// TIA Portal V15.1 export
// export: Created 2024-06-21T08:40:56.7100426Z, ExportSetting WithDefaults, DisplayName Totally Integrated Automation Portal, DisplayVersion V15.1 Update 5, DisplayName TIA Portal Openness, DisplayVersion V15.1 Update 5, DisplayName SINAMICS Startdrive Advanced, DisplayVersion V15.1, DisplayName G130, G150, S120, S150, SINAMICS MV, S210, DisplayVersion V15.1, DisplayName G110M, G120, G120C, G120D, G120P, DisplayVersion V15.1, DisplayName STEP 7 Professional, DisplayVersion V15.1 Update 5, DisplayName STEP 7 Safety, DisplayVersion V15.1, DisplayName WinCC Professional, DisplayVersion V15.1 Update 5, DisplayName SIMATIC Visualization Architect, DisplayVersion V15.1
FUNCTION_BLOCK "L3StopPos"   // FB2188, FBD
TITLE = L3StopPos
{ S7_Optimized_Access := 'TRUE' }
AUTHOR : VCC
FAMILY : Actuator
VERSION : 0.1
// =============================================================================
// This module will be used for a three Position movements.
// It will take care of the Alarms and of the Detections.
// =============================================================================
// stored: AutoNumber false, IsIECCheckEnabled false, IsRetainMemResEnabled false, MemoryReserve 100, SetENOAutomatically False, UDAEnableTagReadback false
   VAR_INPUT
      I_DetPos1 { ExternalAccessible := 'False'; ExternalVisible := 'False'; ExternalWritable := 'False'} : Bool;   // Set detection signal / Pos1 Detection signal
      I_DetPos2 { ExternalAccessible := 'False'; ExternalVisible := 'False'; ExternalWritable := 'False'} : Bool;   // Set detection signal / Pos2 Detection signal
      I_DetPos3 { ExternalAccessible := 'False'; ExternalVisible := 'False'; ExternalWritable := 'False'} : Bool;   // Reset detection signal / Pos3 Detection signal
      I_CmdPos1 { ExternalAccessible := 'False'; ExternalVisible := 'False'; ExternalWritable := 'False'} : Bool;   // function set command / Function Pos1 command
      I_CmdPos2 { ExternalAccessible := 'False'; ExternalVisible := 'False'; ExternalWritable := 'False'} : Bool;   // function set command / Function Pos2 command
      I_CmdPos3 { ExternalAccessible := 'False'; ExternalVisible := 'False'; ExternalWritable := 'False'} : Bool;   // Function reset command / Function Pos3 command
      I_RunPos1 { ExternalAccessible := 'False'; ExternalVisible := 'False'; ExternalWritable := 'False'} : Bool;   // Memory that the Set function is busy / Memory that the Pos1 function is busy
      I_RunPos2 { ExternalAccessible := 'False'; ExternalVisible := 'False'; ExternalWritable := 'False'} : Bool;   // Memory that the Set function is busy / Memory that the Pos2 function is busy
      I_RunPos3 { ExternalAccessible := 'False'; ExternalVisible := 'False'; ExternalWritable := 'False'} : Bool;   // Memory that the Reset function is busy / Memory that the Pos3 function is busy
      I_Pos1IntlkOK { ExternalAccessible := 'False'; ExternalVisible := 'False'; ExternalWritable := 'False'} : Bool;   // Set Interlock / Pos1 Interlock
      I_Pos2IntlkOK { ExternalAccessible := 'False'; ExternalVisible := 'False'; ExternalWritable := 'False'} : Bool;   // Set Interlock / Pos2 Interlock
      I_Pos3IntlkOK { ExternalAccessible := 'False'; ExternalVisible := 'False'; ExternalWritable := 'False'} : Bool;   // Reset Interlock / Pos3 Interlock
      I_SafetyOk { ExternalAccessible := 'False'; ExternalVisible := 'False'; ExternalWritable := 'False'} : Bool;   // Safety Ok
      I_AlarmResetPB { ExternalAccessible := 'False'; ExternalVisible := 'False'; ExternalWritable := 'False'} : Bool := TRUE;   // alarm reset Push Button is activated / Alarm Reset Push Button is Activated
      C_KeepPosition { ExternalAccessible := 'False'; ExternalVisible := 'False'; ExternalWritable := 'False'} : Bool;   // If true, the last position shall be kept ON and checked / If true, the last Position shall be kept ON and checked
      C_EnAlmDet { ExternalAccessible := 'False'; ExternalVisible := 'False'; ExternalWritable := 'False'} : Bool;   // Enable alarm / Enable Alarm
      C_AlarmResetUsed { ExternalAccessible := 'False'; ExternalVisible := 'False'; ExternalWritable := 'False'} : Bool;   // If true, the alarms will be stored untill reseted / If true, the Alarms will be stored untill Reseted
      C_EnAlmOvertime { ExternalAccessible := 'False'; ExternalVisible := 'False'; ExternalWritable := 'False'} : Bool := TRUE;   // Enable Overtime Alarm
      C_RunTimeMaxPos1Warn { ExternalAccessible := 'False'; ExternalVisible := 'False'; ExternalWritable := 'False'} : DInt;   // Maximum Time (ms) that the function may run (create overtime) / Maximum Time (ms) that the function may run (create Overtime)
      C_RunTimeMaxPos1Alm { ExternalAccessible := 'False'; ExternalVisible := 'False'; ExternalWritable := 'False'} : DInt;   // Maximum Time (ms) that the function may run (create overtime) / Maximum Time (ms) that the function may run (create Overtime)
      C_RunTimeMaxPos2Warn { ExternalAccessible := 'False'; ExternalVisible := 'False'; ExternalWritable := 'False'} : DInt;   // Maximum Time (ms) that the function may run (create overtime) / Maximum Time (ms) that the function may run (create Overtime)
      C_RunTimeMaxPos2Alm { ExternalAccessible := 'False'; ExternalVisible := 'False'; ExternalWritable := 'False'} : DInt;   // Maximum Time (ms) that the function may run (create overtime) / Maximum Time (ms) that the function may run (create Overtime)
      C_RunTimeMaxPos3Warn { ExternalAccessible := 'False'; ExternalVisible := 'False'; ExternalWritable := 'False'} : DInt;   // Maximum Time (ms) that the function may run (create overtime) / Maximum Time (ms) that the function may run (create Overtime)
      C_RunTimeMaxPos3Alm { ExternalAccessible := 'False'; ExternalVisible := 'False'; ExternalWritable := 'False'} : DInt;   // Maximum Time (ms) that the function may run (create overtime) / Maximum Time (ms) that the function may run (create Overtime)
      C_TimeAlmFilt { ExternalAccessible := 'False'; ExternalVisible := 'False'; ExternalWritable := 'False'} : DInt := L#2000;   // timer before any actuator alarm will be active (welding..) / timer before any actuator Alarm will be active (welding..)
      C_AlarmSeverityAB { ExternalAccessible := 'False'; ExternalVisible := 'False'; ExternalWritable := 'False'} : Bool;   // Alarm severity
   END_VAR
   VAR_OUTPUT
      O_Pos1 { ExternalAccessible := 'False'; ExternalVisible := 'False'; ExternalWritable := 'False'} : Bool;   // Actuator is in set position / Actuator is in Pos1 Position
      O_Pos2 { ExternalAccessible := 'False'; ExternalVisible := 'False'; ExternalWritable := 'False'} : Bool;   // Actuator is in reset position / Actuator is in Pos2 Position
      O_Pos3 { ExternalAccessible := 'False'; ExternalVisible := 'False'; ExternalWritable := 'False'} : Bool;   // Actuator is in reset position / Actuator is in Pos3 Position
      O_KeepPosPos1Alm { ExternalAccessible := 'False'; ExternalVisible := 'False'; ExternalWritable := 'False'} : Bool;   // Detection Set alarm / Detection Pos1 Alarm
      O_KeepPosPos2Alm { ExternalAccessible := 'False'; ExternalVisible := 'False'; ExternalWritable := 'False'} : Bool;   // Detection Reset alarm / Detection Pos2 Alarm
      O_KeepPosPos3Alm { ExternalAccessible := 'False'; ExternalVisible := 'False'; ExternalWritable := 'False'} : Bool;   // Detection Reset alarm / Detection Pos3 Alarm
      O_MoreThenOneDetAlm { ExternalAccessible := 'False'; ExternalVisible := 'False'; ExternalWritable := 'False'} : Bool;   // Fault condition Both detections ON at the same time / Fault condition More Than One Detections On at the same time
      O_OvtPos1Warn { ExternalAccessible := 'False'; ExternalVisible := 'False'; ExternalWritable := 'False'} : Bool;   // Warning Overtime Set / Warning Overtime Pos1
      O_OvtPos2Warn { ExternalAccessible := 'False'; ExternalVisible := 'False'; ExternalWritable := 'False'} : Bool;   // Warning Overtime Set / Warning Overtime Pos2
      O_OvtPos3Warn { ExternalAccessible := 'False'; ExternalVisible := 'False'; ExternalWritable := 'False'} : Bool;   // Warning Overtime Reset / Warning Overtime Pos3
      O_OvtPos1Alm { ExternalAccessible := 'False'; ExternalVisible := 'False'; ExternalWritable := 'False'} : Bool;   // Alarm Overtime Set / Alarm Overtime Pos1
      O_OvtPos2Alm { ExternalAccessible := 'False'; ExternalVisible := 'False'; ExternalWritable := 'False'} : Bool;   // Alarm Overtime Set / Alarm Overtime Pos2
      O_OvtPos3Alm { ExternalAccessible := 'False'; ExternalVisible := 'False'; ExternalWritable := 'False'} : Bool;   // Alarm Overtime Reset / Alarm Overtime Pos3
      O_ConfigCalibrationAlm { ExternalAccessible := 'False'; ExternalVisible := 'False'; ExternalWritable := 'False'} : Bool;   // Alarm Config/Calibration
      O_CalibrationWarn { ExternalAccessible := 'False'; ExternalVisible := 'False'; ExternalWritable := 'False'} : Bool;   // Warning Calibration
      O_AlarmABCondition { ExternalAccessible := 'False'; ExternalVisible := 'False'; ExternalWritable := 'False'} : Bool;   // Alarm AB condition / Alarm AB Condition
      H_IAnim { ExternalAccessible := 'False'; ExternalVisible := 'False'; ExternalWritable := 'False'} : DWord;   // Icon animation Word / Icon Animation
   END_VAR
   VAR_IN_OUT
      IO_Modes : "Modes";   // Modes
      H_3StopPos : "H_3StopPos";   // Animation
   END_VAR
   VAR
      AlarmReset { ExternalAccessible := 'False'; ExternalVisible := 'False'; ExternalWritable := 'False'} : Bool;   // Alarm Reset Memory
      Pos1PosReq { ExternalAccessible := 'False'; ExternalVisible := 'False'; ExternalWritable := 'False'} : Bool;   // Memorisation of the last set movement / Memorisation of the last Pos1 movement
      Pos2PosReq { ExternalAccessible := 'False'; ExternalVisible := 'False'; ExternalWritable := 'False'} : Bool;   // Memorisation of the last reset movement / Memorisation of the last Pos2 movement
      Pos3PosReq { ExternalAccessible := 'False'; ExternalVisible := 'False'; ExternalWritable := 'False'} : Bool;   // Memorisation of the last reset movement / Memorisation of the last Pos3 movement
      KeepPos1PosOn { ExternalAccessible := 'False'; ExternalVisible := 'False'; ExternalWritable := 'False'} : Bool;   // Check that Set detection is keept on / Check that Pos1 Detection is keept on
      KeepPos2PosOn { ExternalAccessible := 'False'; ExternalVisible := 'False'; ExternalWritable := 'False'} : Bool;   // Check that Set detection is keept on / Check that Pos2 Detection is keept on
      KeepPos3PosOn { ExternalAccessible := 'False'; ExternalVisible := 'False'; ExternalWritable := 'False'} : Bool;   // Check that Set detection is keept on / Check that Pos3 Detection is keept on
      KeepPosPos1StartTimer { ExternalAccessible := 'False'; ExternalVisible := 'False'; ExternalWritable := 'False'} : Bool;   // Detection Set request to start timer / Detection Pos1 Request to start timer
      KeepPosPos2StartTimer { ExternalAccessible := 'False'; ExternalVisible := 'False'; ExternalWritable := 'False'} : Bool;   // Detection Reset request to start timer / Detection Pos2 Request to start timer
      KeepPosPos3StartTimer { ExternalAccessible := 'False'; ExternalVisible := 'False'; ExternalWritable := 'False'} : Bool;   // Detection Reset request to start timer / Detection Pos3 Request to start timer
      MoreThenOneDet { ExternalAccessible := 'False'; ExternalVisible := 'False'; ExternalWritable := 'False'} : Bool;   // Both detections ON at the same time request to start timer / Both Detections ON at the same time Request to start timer
      AlarmFilterStart { ExternalAccessible := 'False'; ExternalVisible := 'False'; ExternalWritable := 'False'} : Bool;   // Alarm filter must be started
      OvtPos1WarnResult { ExternalAccessible := 'False'; ExternalVisible := 'False'; ExternalWritable := 'False'} : Bool;   // Overtime set warning result / Overtime Pos1 warning result
      OvtPos2WarnResult { ExternalAccessible := 'False'; ExternalVisible := 'False'; ExternalWritable := 'False'} : Bool;   // Overtime set warning result / Overtime Pos2 warning result
      OvtPos3WarnResult { ExternalAccessible := 'False'; ExternalVisible := 'False'; ExternalWritable := 'False'} : Bool;   // Overtime reset warning result / Overtime Pos3 warning result
      OvtPos1AlmResult { ExternalAccessible := 'False'; ExternalVisible := 'False'; ExternalWritable := 'False'} : Bool;   // Overtime set alarm result / Overtime Pos1 Alarm result
      OvtPos2AlmResult { ExternalAccessible := 'False'; ExternalVisible := 'False'; ExternalWritable := 'False'} : Bool;   // Overtime reset alarm result / Overtime Pos2 Alarm result
      OvtPos3AlmResult { ExternalAccessible := 'False'; ExternalVisible := 'False'; ExternalWritable := 'False'} : Bool;   // Overtime reset alarm result / Overtime Pos3 Alarm result
      AlmFilterResult { ExternalAccessible := 'False'; ExternalVisible := 'False'; ExternalWritable := 'False'} : Bool;   // Alarm filter result
      MoreThenOneDetAlm { ExternalAccessible := 'False'; ExternalVisible := 'False'; ExternalWritable := 'False'} : Bool;   // Two detection alarm / Pos1 Pos2 Pos3 More Than One Activated
      KeepPos3Alm { ExternalAccessible := 'False'; ExternalVisible := 'False'; ExternalWritable := 'False'} : Bool;   // Keep position Reset alarm / Alarm Keep Position Pos3 Position / Larm Positionsövervakning Pos3 Läge
      KeepPos2Alm { ExternalAccessible := 'False'; ExternalVisible := 'False'; ExternalWritable := 'False'} : Bool;   // Keep position Set alarm / Alarm Keep Position Pos2 Position / Larm Positionsövervakning Pos2 Läge
      KeepPos1Alm { ExternalAccessible := 'False'; ExternalVisible := 'False'; ExternalWritable := 'False'} : Bool;   // Keep position Set alarm / Alarm Keep Position Pos1 Position / Larm Positionsövervakning Pos1 Läge
      OvtPos3Alm { ExternalAccessible := 'False'; ExternalVisible := 'False'; ExternalWritable := 'False'} : Bool;   // Overtime Reset alarm / Overtime Pos3 Alarm
      OvtPos2Alm { ExternalAccessible := 'False'; ExternalVisible := 'False'; ExternalWritable := 'False'} : Bool;   // Overtime Set alarm / Overtime Pos2 Alarm
      OvtPos1Alm { ExternalAccessible := 'False'; ExternalVisible := 'False'; ExternalWritable := 'False'} : Bool;   // Overtime Set alarm / Overtime Pos1 Alarm
      OvtPos3Warn { ExternalAccessible := 'False'; ExternalVisible := 'False'; ExternalWritable := 'False'} : Bool;   // Overtime Reset warning / Overtime Pos3 warning
      OvtPos2Warn { ExternalAccessible := 'False'; ExternalVisible := 'False'; ExternalWritable := 'False'} : Bool;   // Overtime Reset warning / Overtime Pos2 warning
      OvtPos1Warn { ExternalAccessible := 'False'; ExternalVisible := 'False'; ExternalWritable := 'False'} : Bool;   // Overtime Set warning / Overtime Pos1 warning
      ConfigCalibrationAlm { ExternalAccessible := 'False'; ExternalVisible := 'False'; ExternalWritable := 'False'} : Bool;   // Config/Calibration Alarm
      CalibrationWarn { ExternalAccessible := 'False'; ExternalVisible := 'False'; ExternalWritable := 'False'} : Bool;   // Warning Calibration
      Pos1Pos { ExternalAccessible := 'False'; ExternalVisible := 'False'; ExternalWritable := 'False'} : Bool;   // Set position / Pos1 Position
      Pos2Pos { ExternalAccessible := 'False'; ExternalVisible := 'False'; ExternalWritable := 'False'} : Bool;   // Set position / Pos2 Position
      Pos3Pos { ExternalAccessible := 'False'; ExternalVisible := 'False'; ExternalWritable := 'False'} : Bool;   // Reset position / Pos3 Position
      KeepPosPos3AlmCond { ExternalAccessible := 'False'; ExternalVisible := 'False'; ExternalWritable := 'False'} : Bool;   // Keep position reset alarm condition / Keep Position Pos3 Alarm condition
      KeepPosPos2AlmCond { ExternalAccessible := 'False'; ExternalVisible := 'False'; ExternalWritable := 'False'} : Bool;   // Keep position set alarm condition / Keep Position Pos1 Alarm condition
      KeepPosPos1AlmCond { ExternalAccessible := 'False'; ExternalVisible := 'False'; ExternalWritable := 'False'} : Bool;   // Keep position set alarm condition / Keep Position Pos1 Alarm condition
      TwoDetAlmCond { ExternalAccessible := 'False'; ExternalVisible := 'False'; ExternalWritable := 'False'} : Bool;   // Two detector alarm condition / Two or More Detection Alarm condition
      OvtPos3AlmCond { ExternalAccessible := 'False'; ExternalVisible := 'False'; ExternalWritable := 'False'} : Bool;   // Overtime reset alarm condition / Overtime Pos3 Alarm condition
      OvtPos2AlmCond { ExternalAccessible := 'False'; ExternalVisible := 'False'; ExternalWritable := 'False'} : Bool;   // Overtime reset alarm condition / Overtime Pos2 Alarm condition
      OvtPos1AlmCond { ExternalAccessible := 'False'; ExternalVisible := 'False'; ExternalWritable := 'False'} : Bool;   // Overtime set alarm condition / Overtime Pos1 Alarm condition
      Edge { ExternalAccessible := 'False'; ExternalVisible := 'False'; ExternalWritable := 'False'} : Array[1..8] of Bool;   // Edge
      AlarmTimer { ExternalAccessible := 'False'; ExternalVisible := 'False'; ExternalWritable := 'False'} : "LTimer";   // FB
      OvtPos1WarnTimer { ExternalAccessible := 'False'; ExternalVisible := 'False'; ExternalWritable := 'False'} : "LTimer";   // FB
      OvtPos2WarnTimer { ExternalAccessible := 'False'; ExternalVisible := 'False'; ExternalWritable := 'False'} : "LTimer";   // FB
      OvtPos3WarnTimer { ExternalAccessible := 'False'; ExternalVisible := 'False'; ExternalWritable := 'False'} : "LTimer";   // FB
      OvtPos1AlmTimer { ExternalAccessible := 'False'; ExternalVisible := 'False'; ExternalWritable := 'False'} : "LTimer";   // FB
      OvtPos2AlmTimer { ExternalAccessible := 'False'; ExternalVisible := 'False'; ExternalWritable := 'False'} : "LTimer";   // FB
      OvtPos3AlmTimer { ExternalAccessible := 'False'; ExternalVisible := 'False'; ExternalWritable := 'False'} : "LTimer";   // FB
   END_VAR
   VAR RETAIN
      OvtWarnPos1 { ExternalAccessible := 'False'; ExternalVisible := 'False'; ExternalWritable := 'False'} : DInt;   // Alarm Value
      OvtWarnPos2 { ExternalAccessible := 'False'; ExternalVisible := 'False'; ExternalWritable := 'False'} : DInt;   // Alarm Value
      OvtWarnPos3 { ExternalAccessible := 'False'; ExternalVisible := 'False'; ExternalWritable := 'False'} : DInt;   // Alarm Value
      OvtWarnPos1toPos2 { ExternalAccessible := 'False'; ExternalVisible := 'False'; ExternalWritable := 'False'} : DInt;   // Alarm Value
      OvtWarnPos1toPos3 { ExternalAccessible := 'False'; ExternalVisible := 'False'; ExternalWritable := 'False'} : DInt;   // Alarm Value
      OvtWarnPos2toPos3 { ExternalAccessible := 'False'; ExternalVisible := 'False'; ExternalWritable := 'False'} : DInt;   // Alarm Value
      OvtWarnPos2toPos1 { ExternalAccessible := 'False'; ExternalVisible := 'False'; ExternalWritable := 'False'} : DInt;   // Alarm Value
      OvtWarnPos3toPos2 { ExternalAccessible := 'False'; ExternalVisible := 'False'; ExternalWritable := 'False'} : DInt;   // Alarm Value
      OvtWarnPos3toPos1 { ExternalAccessible := 'False'; ExternalVisible := 'False'; ExternalWritable := 'False'} : DInt;   // Alarm Value
      OvtAlarmPos1 { ExternalAccessible := 'False'; ExternalVisible := 'False'; ExternalWritable := 'False'} : DInt;   // Alarm Value
      OvtAlarmPos2 { ExternalAccessible := 'False'; ExternalVisible := 'False'; ExternalWritable := 'False'} : DInt;   // Alarm Value
      OvtAlarmPos3 { ExternalAccessible := 'False'; ExternalVisible := 'False'; ExternalWritable := 'False'} : DInt;   // Alarm Value
      OvtAlarmPos1toPos2 { ExternalAccessible := 'False'; ExternalVisible := 'False'; ExternalWritable := 'False'} : DInt;   // Alarm Value
      OvtAlarmPos1toPos3 { ExternalAccessible := 'False'; ExternalVisible := 'False'; ExternalWritable := 'False'} : DInt;   // Alarm Value
      OvtAlarmPos2toPos3 { ExternalAccessible := 'False'; ExternalVisible := 'False'; ExternalWritable := 'False'} : DInt;   // Alarm Value
      OvtAlarmPos2toPos1 { ExternalAccessible := 'False'; ExternalVisible := 'False'; ExternalWritable := 'False'} : DInt;   // Alarm Value
      OvtAlarmPos3toPos2 { ExternalAccessible := 'False'; ExternalVisible := 'False'; ExternalWritable := 'False'} : DInt;   // Alarm Value
      OvtAlarmPos3toPos1 { ExternalAccessible := 'False'; ExternalVisible := 'False'; ExternalWritable := 'False'} : DInt;   // Alarm Value
      CalibratedPos1toPos2 { ExternalAccessible := 'False'; ExternalVisible := 'False'; ExternalWritable := 'False'} : Bool;   // Calibrated Set
      CalibratedPos1toPos3 { ExternalAccessible := 'False'; ExternalVisible := 'False'; ExternalWritable := 'False'} : Bool;   // Calibrated Reset
      CalibratedPos2toPos3 { ExternalAccessible := 'False'; ExternalVisible := 'False'; ExternalWritable := 'False'} : Bool;   // Calibrated Reset
      CalibratedPos2toPos1 { ExternalAccessible := 'False'; ExternalVisible := 'False'; ExternalWritable := 'False'} : Bool;   // Calibrated Reset
      CalibratedPos3toPos2 { ExternalAccessible := 'False'; ExternalVisible := 'False'; ExternalWritable := 'False'} : Bool;   // Calibrated Reset
      CalibratedPos3toPos1 { ExternalAccessible := 'False'; ExternalVisible := 'False'; ExternalWritable := 'False'} : Bool;   // Calibrated Reset
      MovementPos1toPos3 { ExternalAccessible := 'False'; ExternalVisible := 'False'; ExternalWritable := 'False'} : Bool;   // Calibrated Set
      MovementPos1toPos2 { ExternalAccessible := 'False'; ExternalVisible := 'False'; ExternalWritable := 'False'} : Bool;   // Calibrated Set
      MovementPos3toPos1 { ExternalAccessible := 'False'; ExternalVisible := 'False'; ExternalWritable := 'False'} : Bool;   // Calibrated Set
      MovementPos3toPos2 { ExternalAccessible := 'False'; ExternalVisible := 'False'; ExternalWritable := 'False'} : Bool;   // Calibrated Set
      MovementPos2toPos1 { ExternalAccessible := 'False'; ExternalVisible := 'False'; ExternalWritable := 'False'} : Bool;   // Calibrated Set
      MovementPos2toPos3 { ExternalAccessible := 'False'; ExternalVisible := 'False'; ExternalWritable := 'False'} : Bool;   // Calibrated Set
   END_VAR
   VAR
      AlarmTimeWithConfig { ExternalAccessible := 'False'; ExternalVisible := 'False'; ExternalWritable := 'False'} : Bool;
      AlarmTimeWithCalibration { ExternalAccessible := 'False'; ExternalVisible := 'False'; ExternalWritable := 'False'} : Bool;
      AlmFilterTimerValue { ExternalAccessible := 'False'; ExternalVisible := 'False'; ExternalWritable := 'False'} : DInt;
   END_VAR
   VAR_TEMP
      Cnt : Int;   // Temp
      H_CalibratePos1 : Bool;   // HMI Function
      H_CalibratePos2 : Bool;   // HMI Function
      H_CalibratePos3 : Bool;   // HMI Function
      TempReal : Real;
   END_VAR
   VAR_TEMP   // added for the SCL form of the ladder/FBD networks
      _w1 : Bool;
      _w2 : Bool;
      _w3 : Bool;
      _w4 : Bool;
      _w5 : Bool;
      _w6 : Bool;
      _w7 : Bool;
      _w8 : Bool;
      _w9 : Bool;
      _w10 : Bool;
      _w11 : Bool;
      _w12 : Bool;
      _w13 : Bool;
      _w14 : Bool;
      _w15 : Bool;
   END_VAR
BEGIN

REGION Network 1: **** 1 - Inputs **** HMI Commands
   // Extract the Commands from HMIRobCmd / Extract the Commands from HMI
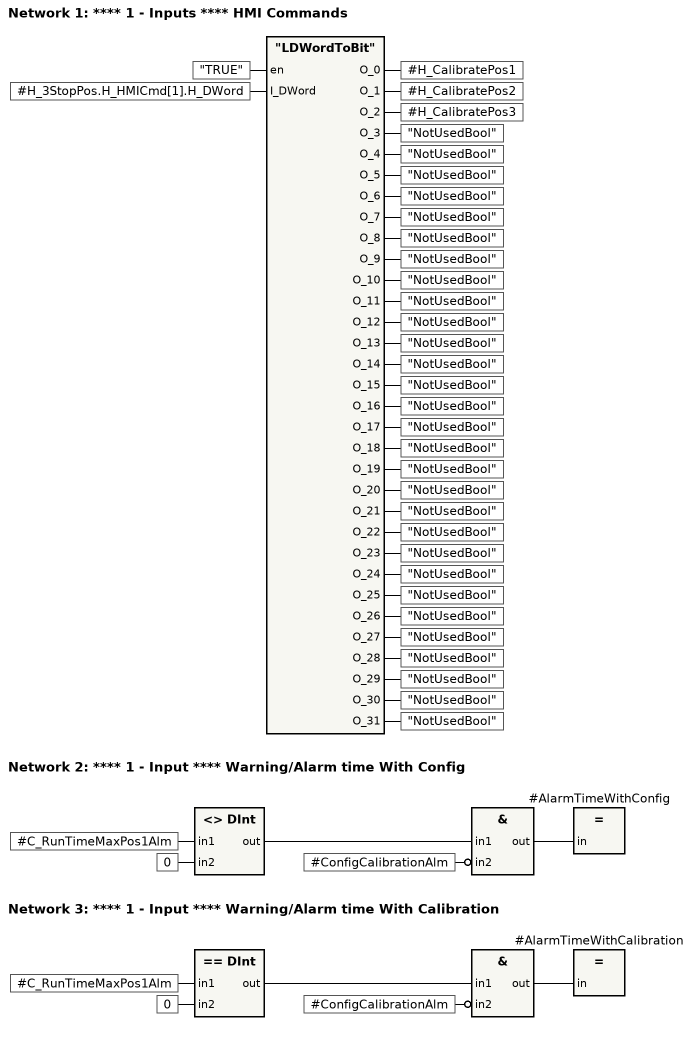
   IF "TRUE" THEN
       "LDWordToBit"(I_DWord := #H_3StopPos.H_HMICmd[1].H_DWord,
                     O_0 => #H_CalibratePos1,
                     O_1 => #H_CalibratePos2,
                     O_2 => #H_CalibratePos3,
                     O_3 => "NotUsedBool",
                     O_4 => "NotUsedBool",
                     O_5 => "NotUsedBool",
                     O_6 => "NotUsedBool",
                     O_7 => "NotUsedBool",
                     O_8 => "NotUsedBool",
                     O_9 => "NotUsedBool",
                     O_10 => "NotUsedBool",
                     O_11 => "NotUsedBool",
                     O_12 => "NotUsedBool",
                     O_13 => "NotUsedBool",
                     O_14 => "NotUsedBool",
                     O_15 => "NotUsedBool",
                     O_16 => "NotUsedBool",
                     O_17 => "NotUsedBool",
                     O_18 => "NotUsedBool",
                     O_19 => "NotUsedBool",
                     O_20 => "NotUsedBool",
                     O_21 => "NotUsedBool",
                     O_22 => "NotUsedBool",
                     O_23 => "NotUsedBool",
                     O_24 => "NotUsedBool",
                     O_25 => "NotUsedBool",
                     O_26 => "NotUsedBool",
                     O_27 => "NotUsedBool",
                     O_28 => "NotUsedBool",
                     O_29 => "NotUsedBool",
                     O_30 => "NotUsedBool",
                     O_31 => "NotUsedBool");
   END_IF;
END_REGION

REGION Network 2: **** 1 - Input **** Warning/Alarm time With Config
   #AlarmTimeWithConfig := (#C_RunTimeMaxPos1Alm <> 0) AND NOT #ConfigCalibrationAlm;
END_REGION

REGION Network 3: **** 1 - Input **** Warning/Alarm time With Calibration
   #AlarmTimeWithCalibration := (#C_RunTimeMaxPos1Alm = 0) AND NOT #ConfigCalibrationAlm;
END_REGION

REGION Network 4: Calibrated Set / **** 1 - Input **** Ovt Values / **** 1 - Inputs **** Ovt Values
   // Ovt Values
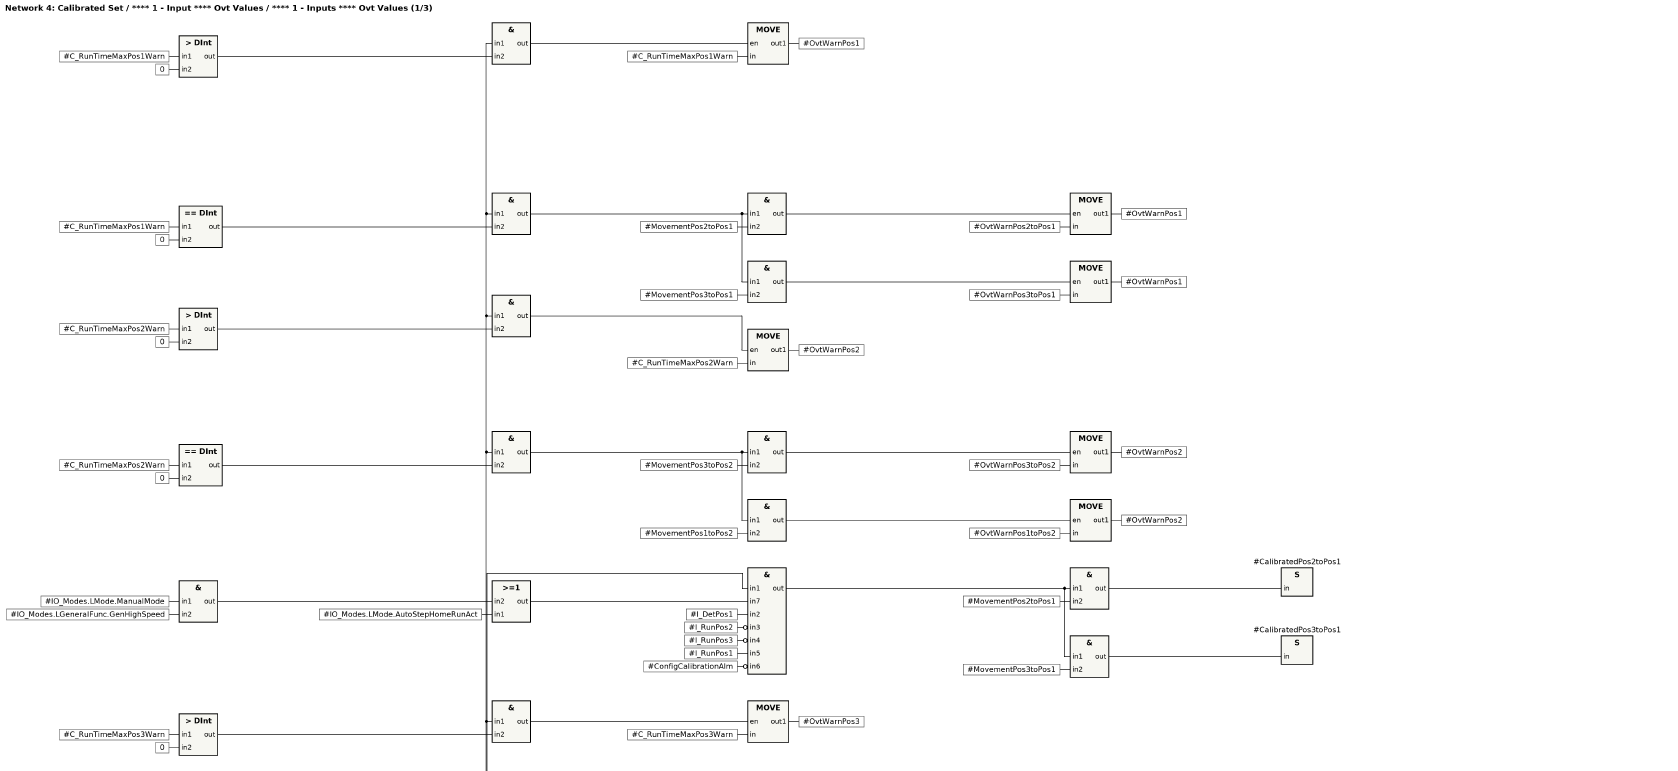
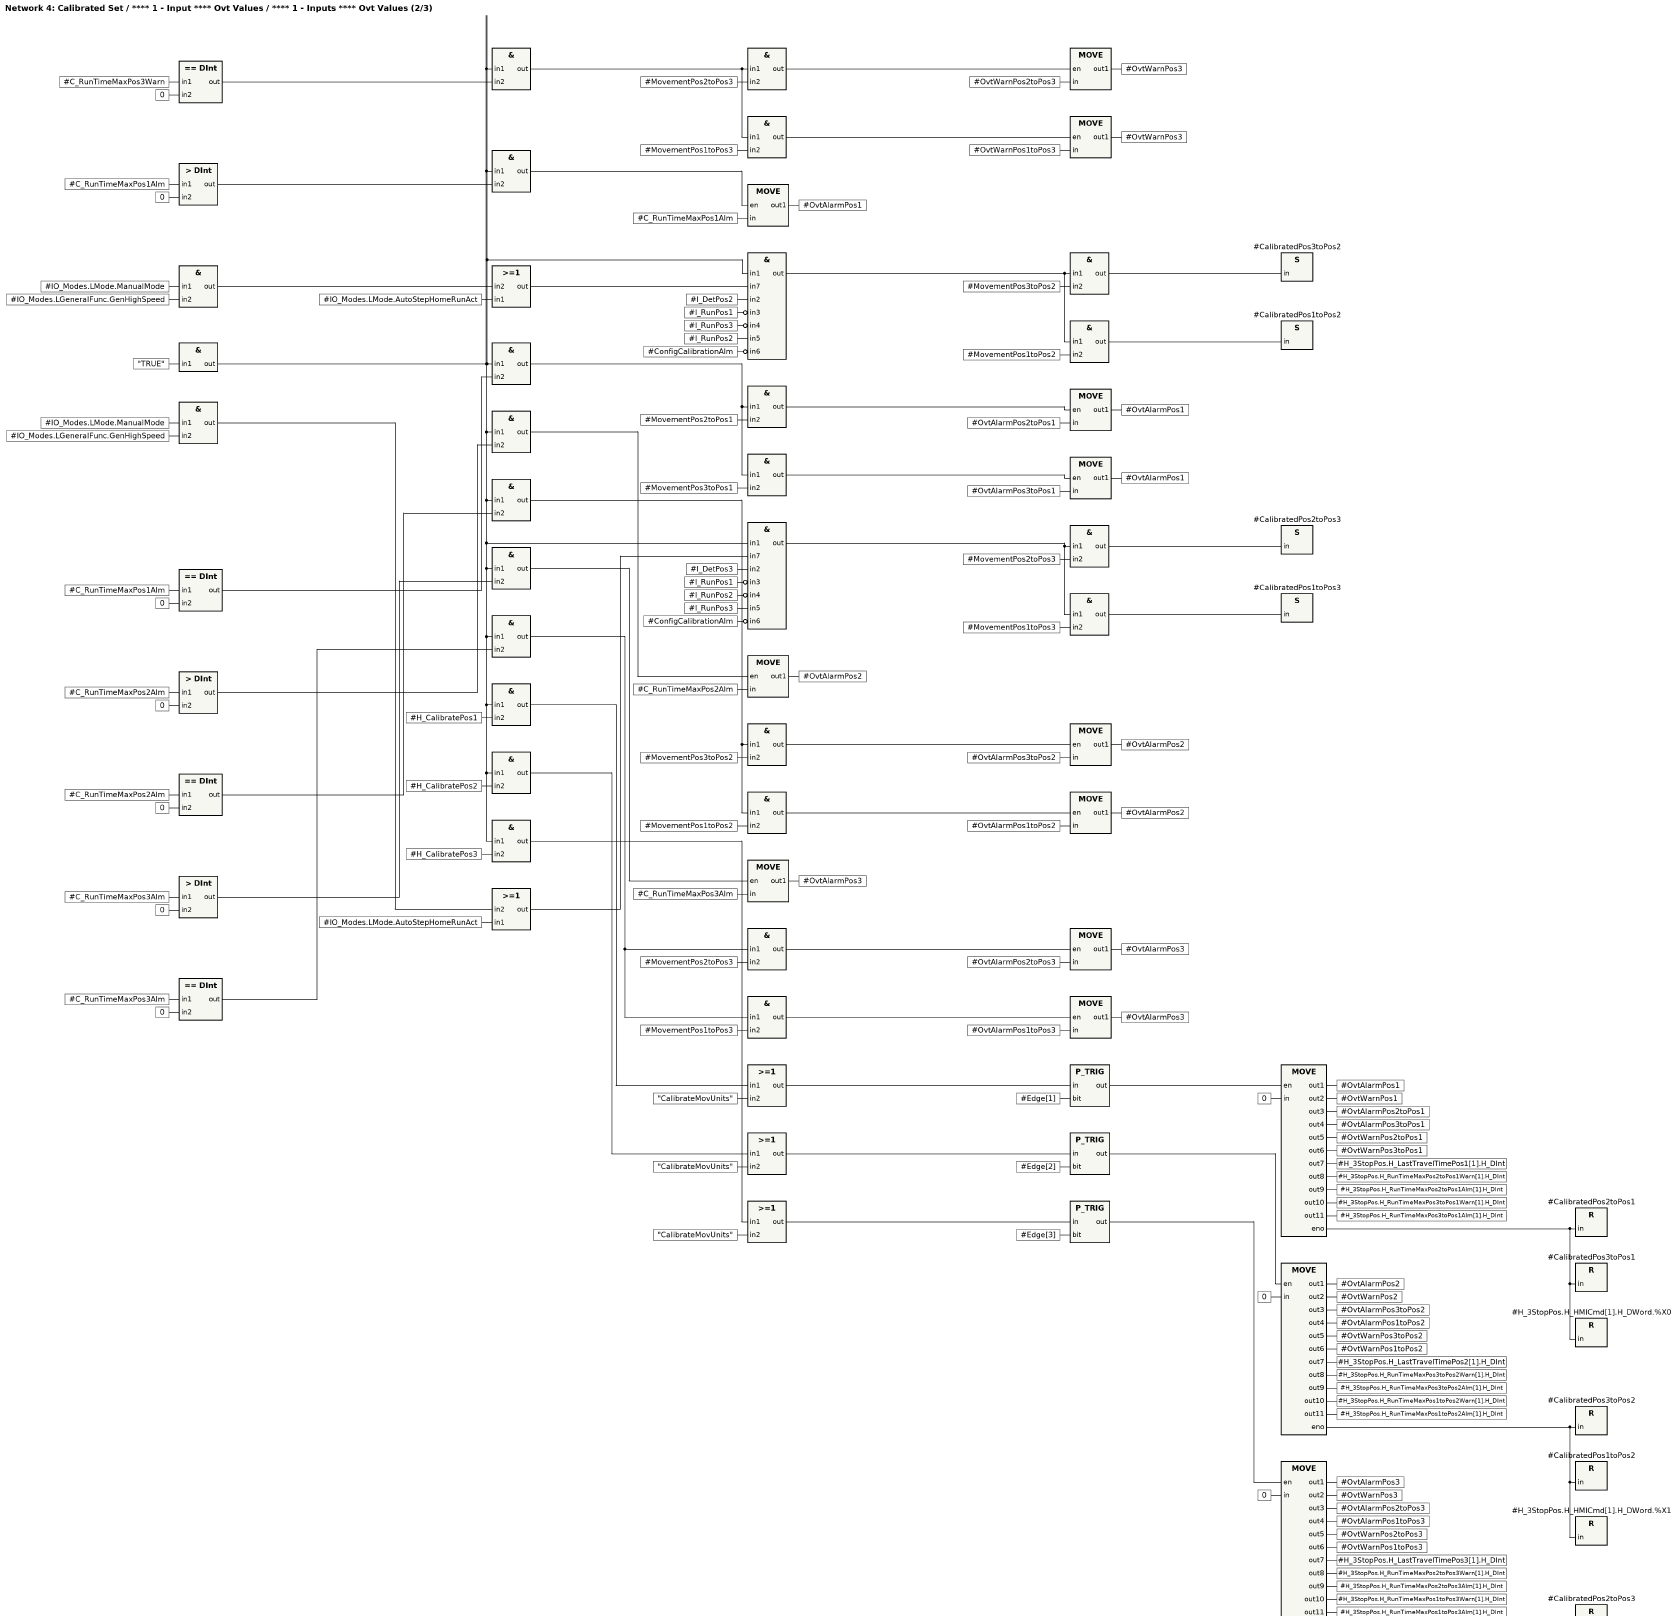
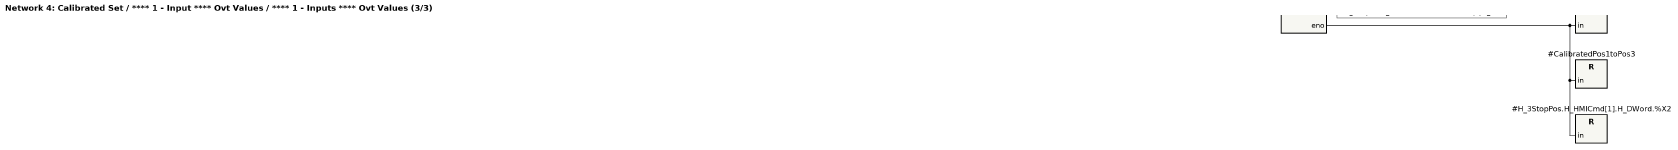
   // ENO of a box is taken as its EN; it also drops when the box reports an error
   IF "TRUE" AND (#C_RunTimeMaxPos1Warn > 0) THEN #OvtWarnPos1 := #C_RunTimeMaxPos1Warn; END_IF;
   #_w1 := "TRUE" AND (#C_RunTimeMaxPos1Warn = 0);
   IF #_w1 AND #MovementPos2toPos1 THEN #OvtWarnPos1 := #OvtWarnPos2toPos1; END_IF;
   IF #_w1 AND #MovementPos3toPos1 THEN #OvtWarnPos1 := #OvtWarnPos3toPos1; END_IF;
   IF "TRUE" AND (#C_RunTimeMaxPos2Warn > 0) THEN #OvtWarnPos2 := #C_RunTimeMaxPos2Warn; END_IF;
   #_w2 := "TRUE" AND (#C_RunTimeMaxPos2Warn = 0);
   IF #_w2 AND #MovementPos3toPos2 THEN #OvtWarnPos2 := #OvtWarnPos3toPos2; END_IF;
   IF #_w2 AND #MovementPos1toPos2 THEN #OvtWarnPos2 := #OvtWarnPos1toPos2; END_IF;
   IF "TRUE" AND (#C_RunTimeMaxPos3Warn > 0) THEN #OvtWarnPos3 := #C_RunTimeMaxPos3Warn; END_IF;
   #_w3 := "TRUE" AND (#C_RunTimeMaxPos3Warn = 0);
   IF #_w3 AND #MovementPos2toPos3 THEN #OvtWarnPos3 := #OvtWarnPos2toPos3; END_IF;
   IF #_w3 AND #MovementPos1toPos3 THEN #OvtWarnPos3 := #OvtWarnPos1toPos3; END_IF;
   IF "TRUE" AND (#C_RunTimeMaxPos1Alm > 0) THEN #OvtAlarmPos1 := #C_RunTimeMaxPos1Alm; END_IF;
   #_w4 := "TRUE" AND (#C_RunTimeMaxPos1Alm = 0);
   IF #_w4 AND #MovementPos2toPos1 THEN #OvtAlarmPos1 := #OvtAlarmPos2toPos1; END_IF;
   IF #_w4 AND #MovementPos3toPos1 THEN #OvtAlarmPos1 := #OvtAlarmPos3toPos1; END_IF;
   IF "TRUE" AND (#C_RunTimeMaxPos2Alm > 0) THEN #OvtAlarmPos2 := #C_RunTimeMaxPos2Alm; END_IF;
   #_w5 := "TRUE" AND (#C_RunTimeMaxPos2Alm = 0);
   IF #_w5 AND #MovementPos3toPos2 THEN #OvtAlarmPos2 := #OvtAlarmPos3toPos2; END_IF;
   IF #_w5 AND #MovementPos1toPos2 THEN #OvtAlarmPos2 := #OvtAlarmPos1toPos2; END_IF;
   IF "TRUE" AND (#C_RunTimeMaxPos3Alm > 0) THEN #OvtAlarmPos3 := #C_RunTimeMaxPos3Alm; END_IF;
   #_w6 := "TRUE" AND (#C_RunTimeMaxPos3Alm = 0);
   IF #_w6 AND #MovementPos2toPos3 THEN #OvtAlarmPos3 := #OvtAlarmPos2toPos3; END_IF;
   IF #_w6 AND #MovementPos1toPos3 THEN #OvtAlarmPos3 := #OvtAlarmPos1toPos3; END_IF;
   #_w7 := "TRUE" AND ((#IO_Modes.LMode.ManualMode AND #IO_Modes.LGeneralFunc.GenHighSpeed) OR #IO_Modes.LMode.AutoStepHomeRunAct) AND #I_DetPos1 AND NOT #I_RunPos2 AND NOT #I_RunPos3 AND #I_RunPos1 AND NOT #ConfigCalibrationAlm;
   IF #_w7 AND #MovementPos2toPos1 THEN #CalibratedPos2toPos1 := TRUE; END_IF;
   IF #_w7 AND #MovementPos3toPos1 THEN #CalibratedPos3toPos1 := TRUE; END_IF;
   #_w8 := "TRUE" AND ((#IO_Modes.LMode.ManualMode AND #IO_Modes.LGeneralFunc.GenHighSpeed) OR #IO_Modes.LMode.AutoStepHomeRunAct) AND #I_DetPos2 AND NOT #I_RunPos1 AND NOT #I_RunPos3 AND #I_RunPos2 AND NOT #ConfigCalibrationAlm;
   IF #_w8 AND #MovementPos3toPos2 THEN #CalibratedPos3toPos2 := TRUE; END_IF;
   IF #_w8 AND #MovementPos1toPos2 THEN #CalibratedPos1toPos2 := TRUE; END_IF;
   #_w9 := "TRUE" AND ((#IO_Modes.LMode.ManualMode AND #IO_Modes.LGeneralFunc.GenHighSpeed) OR #IO_Modes.LMode.AutoStepHomeRunAct) AND #I_DetPos3 AND NOT #I_RunPos1 AND NOT #I_RunPos2 AND #I_RunPos3 AND NOT #ConfigCalibrationAlm;
   IF #_w9 AND #MovementPos2toPos3 THEN #CalibratedPos2toPos3 := TRUE; END_IF;
   IF #_w9 AND #MovementPos1toPos3 THEN #CalibratedPos1toPos3 := TRUE; END_IF;
   #_w10 := ("TRUE" AND #H_CalibratePos1) OR "CalibrateMovUnits";
   #_w11 := #_w10 AND NOT #Edge[1];   // rising edge
   #Edge[1] := #_w10;
   IF #_w11 THEN
       #OvtAlarmPos1 := 0;
       #OvtWarnPos1 := 0;
       #OvtAlarmPos2toPos1 := 0;
       #OvtAlarmPos3toPos1 := 0;
       #OvtWarnPos2toPos1 := 0;
       #OvtWarnPos3toPos1 := 0;
       #H_3StopPos.H_LastTravelTimePos1[1].H_DInt := 0;
       #H_3StopPos.H_RunTimeMaxPos2toPos1Warn[1].H_DInt := 0;
       #H_3StopPos.H_RunTimeMaxPos2toPos1Alm[1].H_DInt := 0;
       #H_3StopPos.H_RunTimeMaxPos3toPos1Warn[1].H_DInt := 0;
       #H_3StopPos.H_RunTimeMaxPos3toPos1Alm[1].H_DInt := 0;
       #CalibratedPos2toPos1 := FALSE;
       #CalibratedPos3toPos1 := FALSE;
       #H_3StopPos.H_HMICmd[1].H_DWord.%X0 := FALSE;
   END_IF;
   #_w12 := ("TRUE" AND #H_CalibratePos2) OR "CalibrateMovUnits";
   #_w13 := #_w12 AND NOT #Edge[2];   // rising edge
   #Edge[2] := #_w12;
   IF #_w13 THEN
       #OvtAlarmPos2 := 0;
       #OvtWarnPos2 := 0;
       #OvtAlarmPos3toPos2 := 0;
       #OvtAlarmPos1toPos2 := 0;
       #OvtWarnPos3toPos2 := 0;
       #OvtWarnPos1toPos2 := 0;
       #H_3StopPos.H_LastTravelTimePos2[1].H_DInt := 0;
       #H_3StopPos.H_RunTimeMaxPos3toPos2Warn[1].H_DInt := 0;
       #H_3StopPos.H_RunTimeMaxPos3toPos2Alm[1].H_DInt := 0;
       #H_3StopPos.H_RunTimeMaxPos1toPos2Warn[1].H_DInt := 0;
       #H_3StopPos.H_RunTimeMaxPos1toPos2Alm[1].H_DInt := 0;
       #CalibratedPos3toPos2 := FALSE;
       #CalibratedPos1toPos2 := FALSE;
       #H_3StopPos.H_HMICmd[1].H_DWord.%X1 := FALSE;
   END_IF;
   #_w14 := ("TRUE" AND #H_CalibratePos3) OR "CalibrateMovUnits";
   #_w15 := #_w14 AND NOT #Edge[3];   // rising edge
   #Edge[3] := #_w14;
   IF #_w15 THEN
       #OvtAlarmPos3 := 0;
       #OvtWarnPos3 := 0;
       #OvtAlarmPos2toPos3 := 0;
       #OvtAlarmPos1toPos3 := 0;
       #OvtWarnPos2toPos3 := 0;
       #OvtWarnPos1toPos3 := 0;
       #H_3StopPos.H_LastTravelTimePos3[1].H_DInt := 0;
       #H_3StopPos.H_RunTimeMaxPos2toPos3Warn[1].H_DInt := 0;
       #H_3StopPos.H_RunTimeMaxPos2toPos3Alm[1].H_DInt := 0;
       #H_3StopPos.H_RunTimeMaxPos1toPos3Warn[1].H_DInt := 0;
       #H_3StopPos.H_RunTimeMaxPos1toPos3Alm[1].H_DInt := 0;
       #CalibratedPos2toPos3 := FALSE;
       #CalibratedPos1toPos3 := FALSE;
       #H_3StopPos.H_HMICmd[1].H_DWord.%X2 := FALSE;
   END_IF;
END_REGION

REGION Network 5: **** 1 - Input **** Start Movement from Pos1 to Pos3
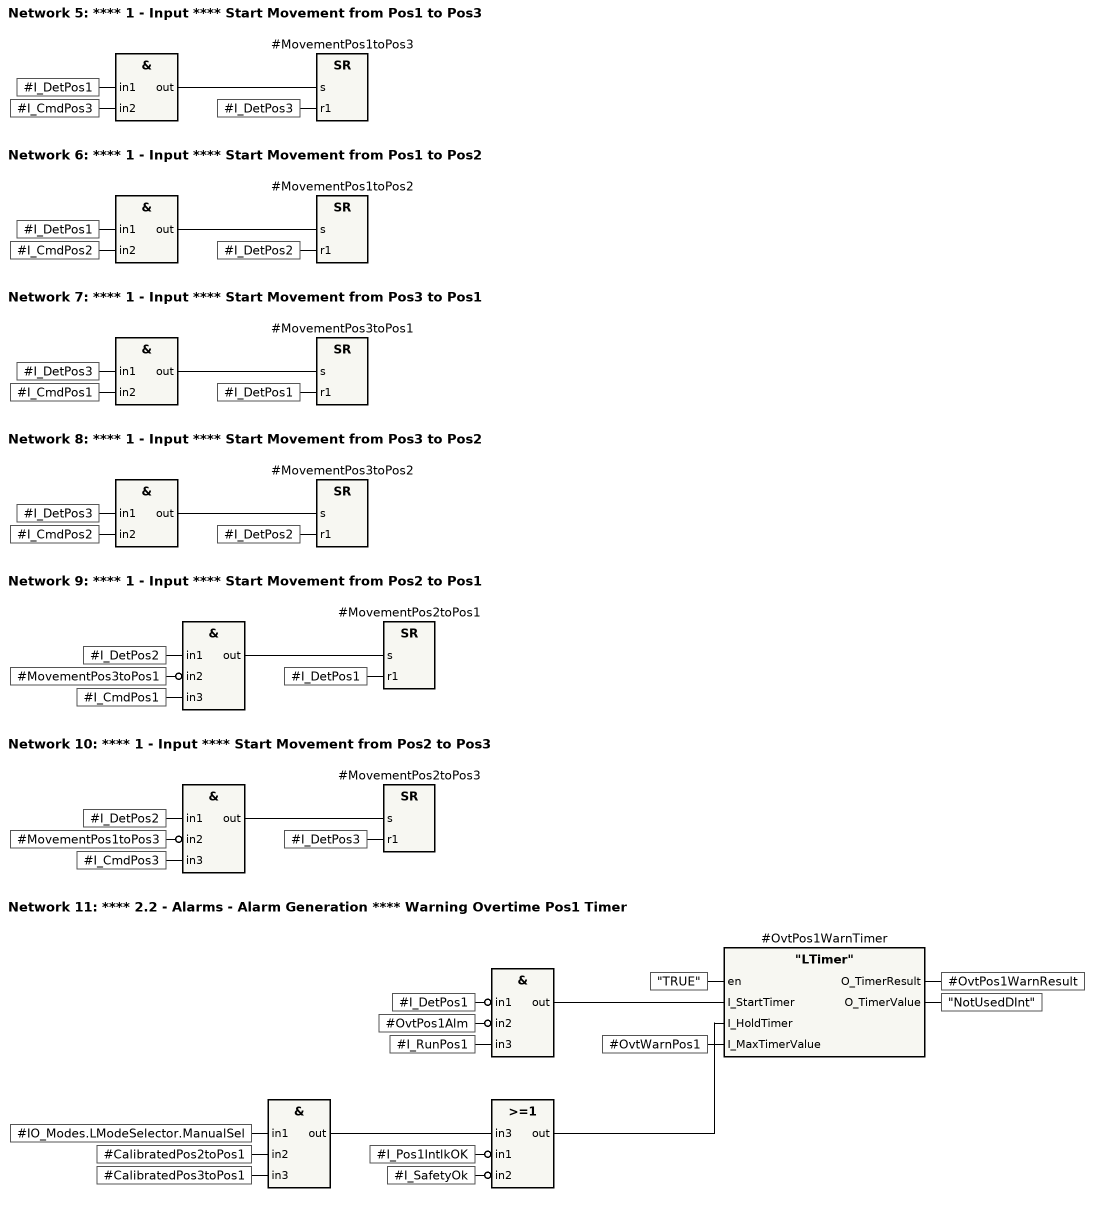
   IF #I_DetPos1 AND #I_CmdPos3 THEN
       #MovementPos1toPos3 := TRUE;   // SR flip-flop
   END_IF;
   IF #I_DetPos3 THEN #MovementPos1toPos3 := FALSE; END_IF;
END_REGION

REGION Network 6: **** 1 - Input **** Start Movement from Pos1 to Pos2
   IF #I_DetPos1 AND #I_CmdPos2 THEN
       #MovementPos1toPos2 := TRUE;   // SR flip-flop
   END_IF;
   IF #I_DetPos2 THEN #MovementPos1toPos2 := FALSE; END_IF;
END_REGION

REGION Network 7: **** 1 - Input **** Start Movement from Pos3 to Pos1
   IF #I_DetPos3 AND #I_CmdPos1 THEN
       #MovementPos3toPos1 := TRUE;   // SR flip-flop
   END_IF;
   IF #I_DetPos1 THEN #MovementPos3toPos1 := FALSE; END_IF;
END_REGION

REGION Network 8: **** 1 - Input **** Start Movement from Pos3 to Pos2
   IF #I_DetPos3 AND #I_CmdPos2 THEN
       #MovementPos3toPos2 := TRUE;   // SR flip-flop
   END_IF;
   IF #I_DetPos2 THEN #MovementPos3toPos2 := FALSE; END_IF;
END_REGION

REGION Network 9: **** 1 - Input **** Start Movement from Pos2 to Pos1
   IF #I_DetPos2 AND NOT #MovementPos3toPos1 AND #I_CmdPos1 THEN
       #MovementPos2toPos1 := TRUE;   // SR flip-flop
   END_IF;
   IF #I_DetPos1 THEN #MovementPos2toPos1 := FALSE; END_IF;
END_REGION

REGION Network 10: **** 1 - Input **** Start Movement from Pos2 to Pos3
   IF #I_DetPos2 AND NOT #MovementPos1toPos3 AND #I_CmdPos3 THEN
       #MovementPos2toPos3 := TRUE;   // SR flip-flop
   END_IF;
   IF #I_DetPos3 THEN #MovementPos2toPos3 := FALSE; END_IF;
END_REGION

REGION Network 11: **** 2.2 - Alarms - Alarm Generation **** Warning Overtime Pos1 Timer
   // Warning Overtime Pos1 Timer
   IF "TRUE" THEN
       #OvtPos1WarnTimer(I_StartTimer := NOT #I_DetPos1 AND NOT #OvtPos1Alm AND #I_RunPos1,   // "LTimer"
                         I_HoldTimer := (#IO_Modes.LModeSelector.ManualSel AND #CalibratedPos2toPos1 AND #CalibratedPos3toPos1) OR NOT #I_Pos1IntlkOK OR NOT #I_SafetyOk,
                         I_MaxTimerValue := #OvtWarnPos1,
                         O_TimerResult => #OvtPos1WarnResult,
                         O_TimerValue => "NotUsedDInt");
   END_IF;
END_REGION

REGION Network 12: **** 2.2 - Alarms - Alarm Generation **** Warning Overtime Pos1 Memorisation
   // Warning Overtime Pos1 Memorisation
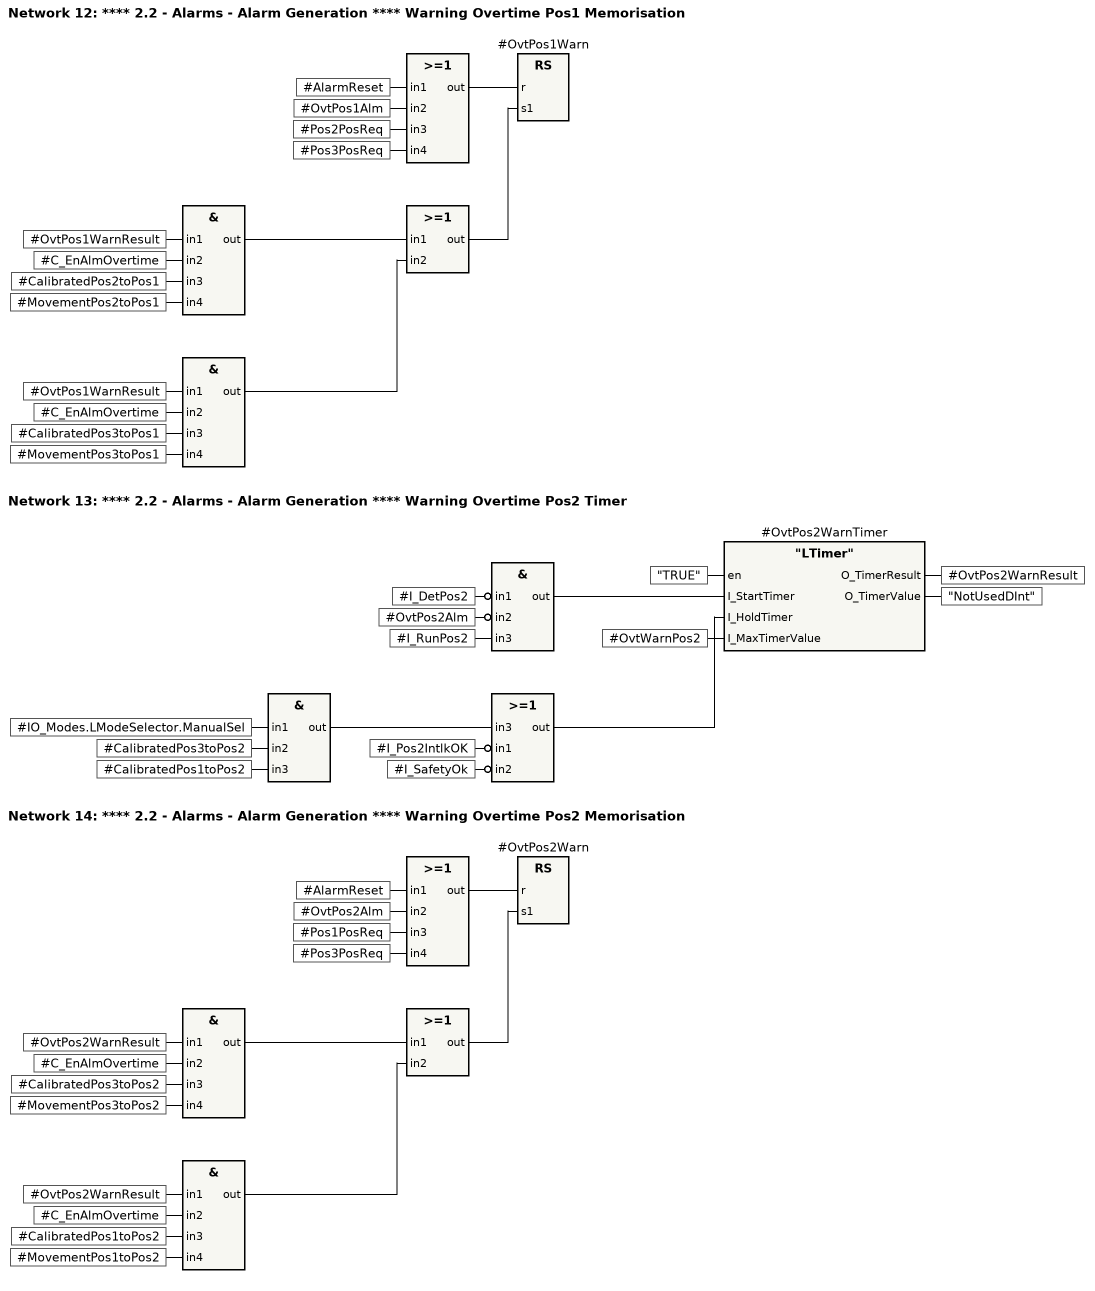
   IF #AlarmReset OR #OvtPos1Alm OR #Pos2PosReq OR #Pos3PosReq THEN
       #OvtPos1Warn := FALSE;   // RS flip-flop
   END_IF;
   IF (#OvtPos1WarnResult AND #C_EnAlmOvertime AND #CalibratedPos2toPos1 AND #MovementPos2toPos1) OR (#OvtPos1WarnResult AND #C_EnAlmOvertime AND #CalibratedPos3toPos1 AND #MovementPos3toPos1) THEN
       #OvtPos1Warn := TRUE;
   END_IF;
END_REGION

REGION Network 13: **** 2.2 - Alarms - Alarm Generation **** Warning Overtime Pos2 Timer
   // Warning Overtime Pos2 Timer
   IF "TRUE" THEN
       #OvtPos2WarnTimer(I_StartTimer := NOT #I_DetPos2 AND NOT #OvtPos2Alm AND #I_RunPos2,   // "LTimer"
                         I_HoldTimer := (#IO_Modes.LModeSelector.ManualSel AND #CalibratedPos3toPos2 AND #CalibratedPos1toPos2) OR NOT #I_Pos2IntlkOK OR NOT #I_SafetyOk,
                         I_MaxTimerValue := #OvtWarnPos2,
                         O_TimerResult => #OvtPos2WarnResult,
                         O_TimerValue => "NotUsedDInt");
   END_IF;
END_REGION

REGION Network 14: **** 2.2 - Alarms - Alarm Generation **** Warning Overtime Pos2 Memorisation
   // Warning Overtime Pos2 Memorisation
   IF #AlarmReset OR #OvtPos2Alm OR #Pos1PosReq OR #Pos3PosReq THEN
       #OvtPos2Warn := FALSE;   // RS flip-flop
   END_IF;
   IF (#OvtPos2WarnResult AND #C_EnAlmOvertime AND #CalibratedPos3toPos2 AND #MovementPos3toPos2) OR (#OvtPos2WarnResult AND #C_EnAlmOvertime AND #CalibratedPos1toPos2 AND #MovementPos1toPos2) THEN
       #OvtPos2Warn := TRUE;
   END_IF;
END_REGION

REGION Network 15: **** 2.2 - Alarms - Alarm Generation **** Warning Overtime Pos3 / **** 2.2 - Alarms - Alarm Generation **** Warning Overtime Pos3 Timer
   // Warning Overtime Pos3
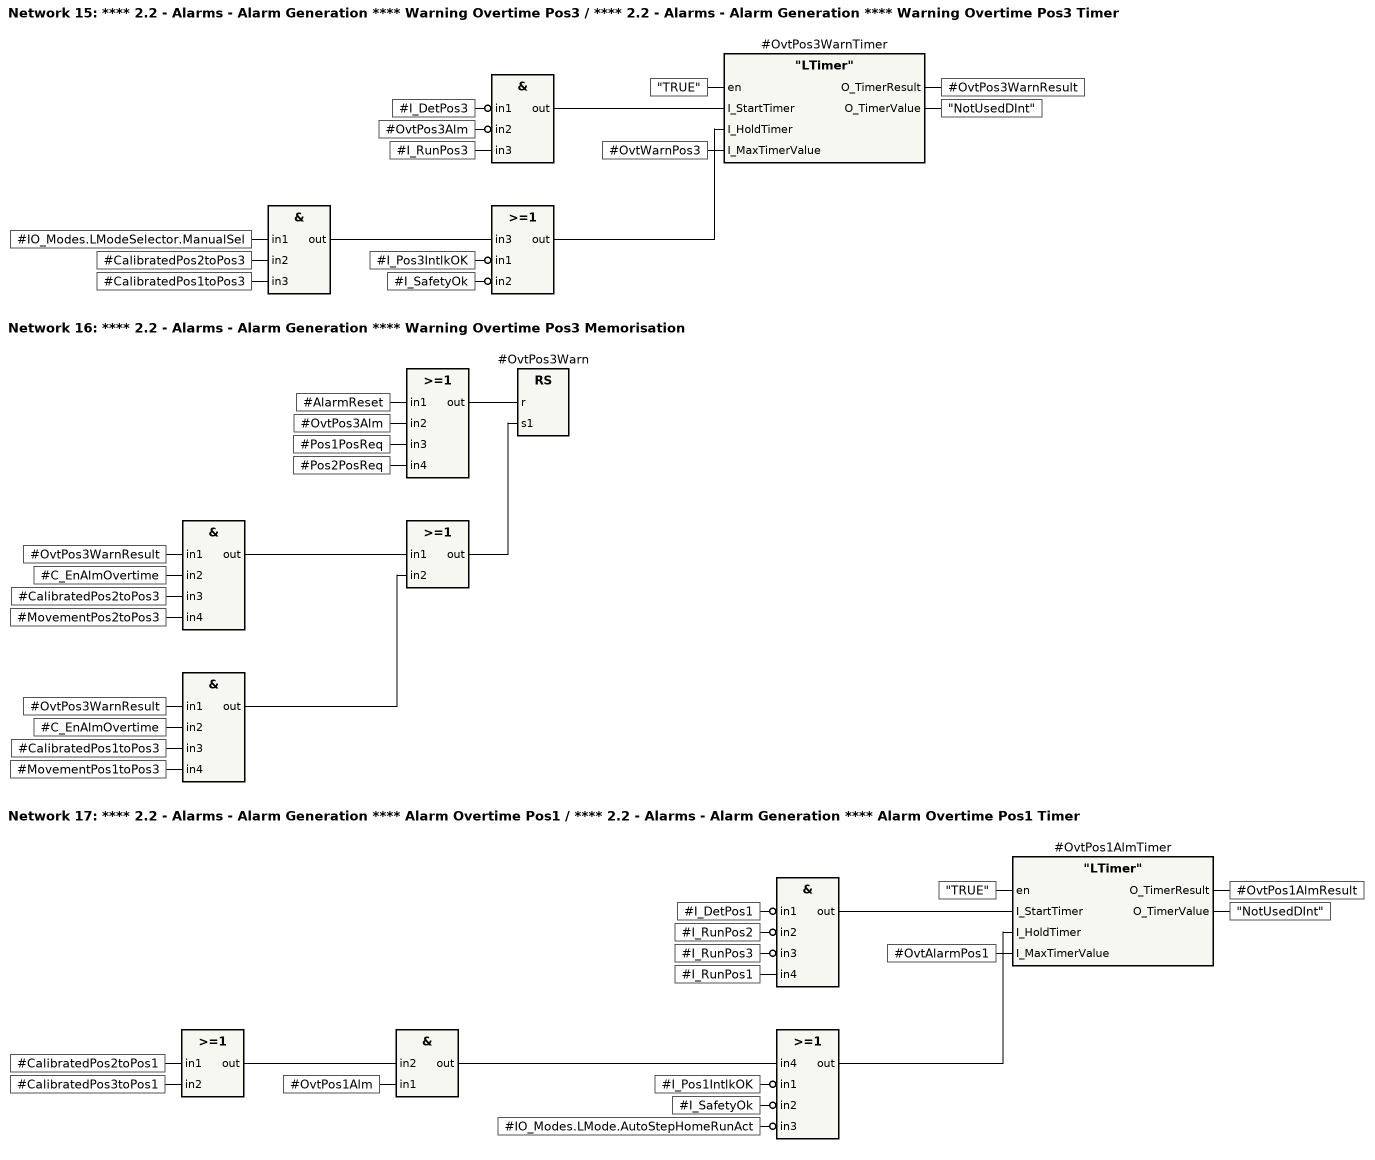
   IF "TRUE" THEN
       #OvtPos3WarnTimer(I_StartTimer := NOT #I_DetPos3 AND NOT #OvtPos3Alm AND #I_RunPos3,   // "LTimer"
                         I_HoldTimer := (#IO_Modes.LModeSelector.ManualSel AND #CalibratedPos2toPos3 AND #CalibratedPos1toPos3) OR NOT #I_Pos3IntlkOK OR NOT #I_SafetyOk,
                         I_MaxTimerValue := #OvtWarnPos3,
                         O_TimerResult => #OvtPos3WarnResult,
                         O_TimerValue => "NotUsedDInt");
   END_IF;
END_REGION

REGION Network 16: **** 2.2 - Alarms - Alarm Generation **** Warning Overtime Pos3 Memorisation
   // Warning Overtime Pos3  Memorisation
   IF #AlarmReset OR #OvtPos3Alm OR #Pos1PosReq OR #Pos2PosReq THEN
       #OvtPos3Warn := FALSE;   // RS flip-flop
   END_IF;
   IF (#OvtPos3WarnResult AND #C_EnAlmOvertime AND #CalibratedPos2toPos3 AND #MovementPos2toPos3) OR (#OvtPos3WarnResult AND #C_EnAlmOvertime AND #CalibratedPos1toPos3 AND #MovementPos1toPos3) THEN
       #OvtPos3Warn := TRUE;
   END_IF;
END_REGION

REGION Network 17: **** 2.2 - Alarms - Alarm Generation **** Alarm Overtime Pos1 / **** 2.2 - Alarms - Alarm Generation **** Alarm Overtime Pos1 Timer
   // Alarm Overtime Pos1
   IF "TRUE" THEN
       #OvtPos1AlmTimer(I_StartTimer := NOT #I_DetPos1 AND NOT #I_RunPos2 AND NOT #I_RunPos3 AND #I_RunPos1,   // "LTimer"
                        I_HoldTimer := ((#CalibratedPos2toPos1 OR #CalibratedPos3toPos1) AND #OvtPos1Alm) OR NOT #I_Pos1IntlkOK OR NOT #I_SafetyOk OR NOT #IO_Modes.LMode.AutoStepHomeRunAct,
                        I_MaxTimerValue := #OvtAlarmPos1,
                        O_TimerResult => #OvtPos1AlmResult,
                        O_TimerValue => "NotUsedDInt");
   END_IF;
END_REGION

REGION Network 18: **** 2.2 - Alarms - Alarm Generation **** Alarm Overtime Pos1 Timer -- Calculation Warning/Alarm Time
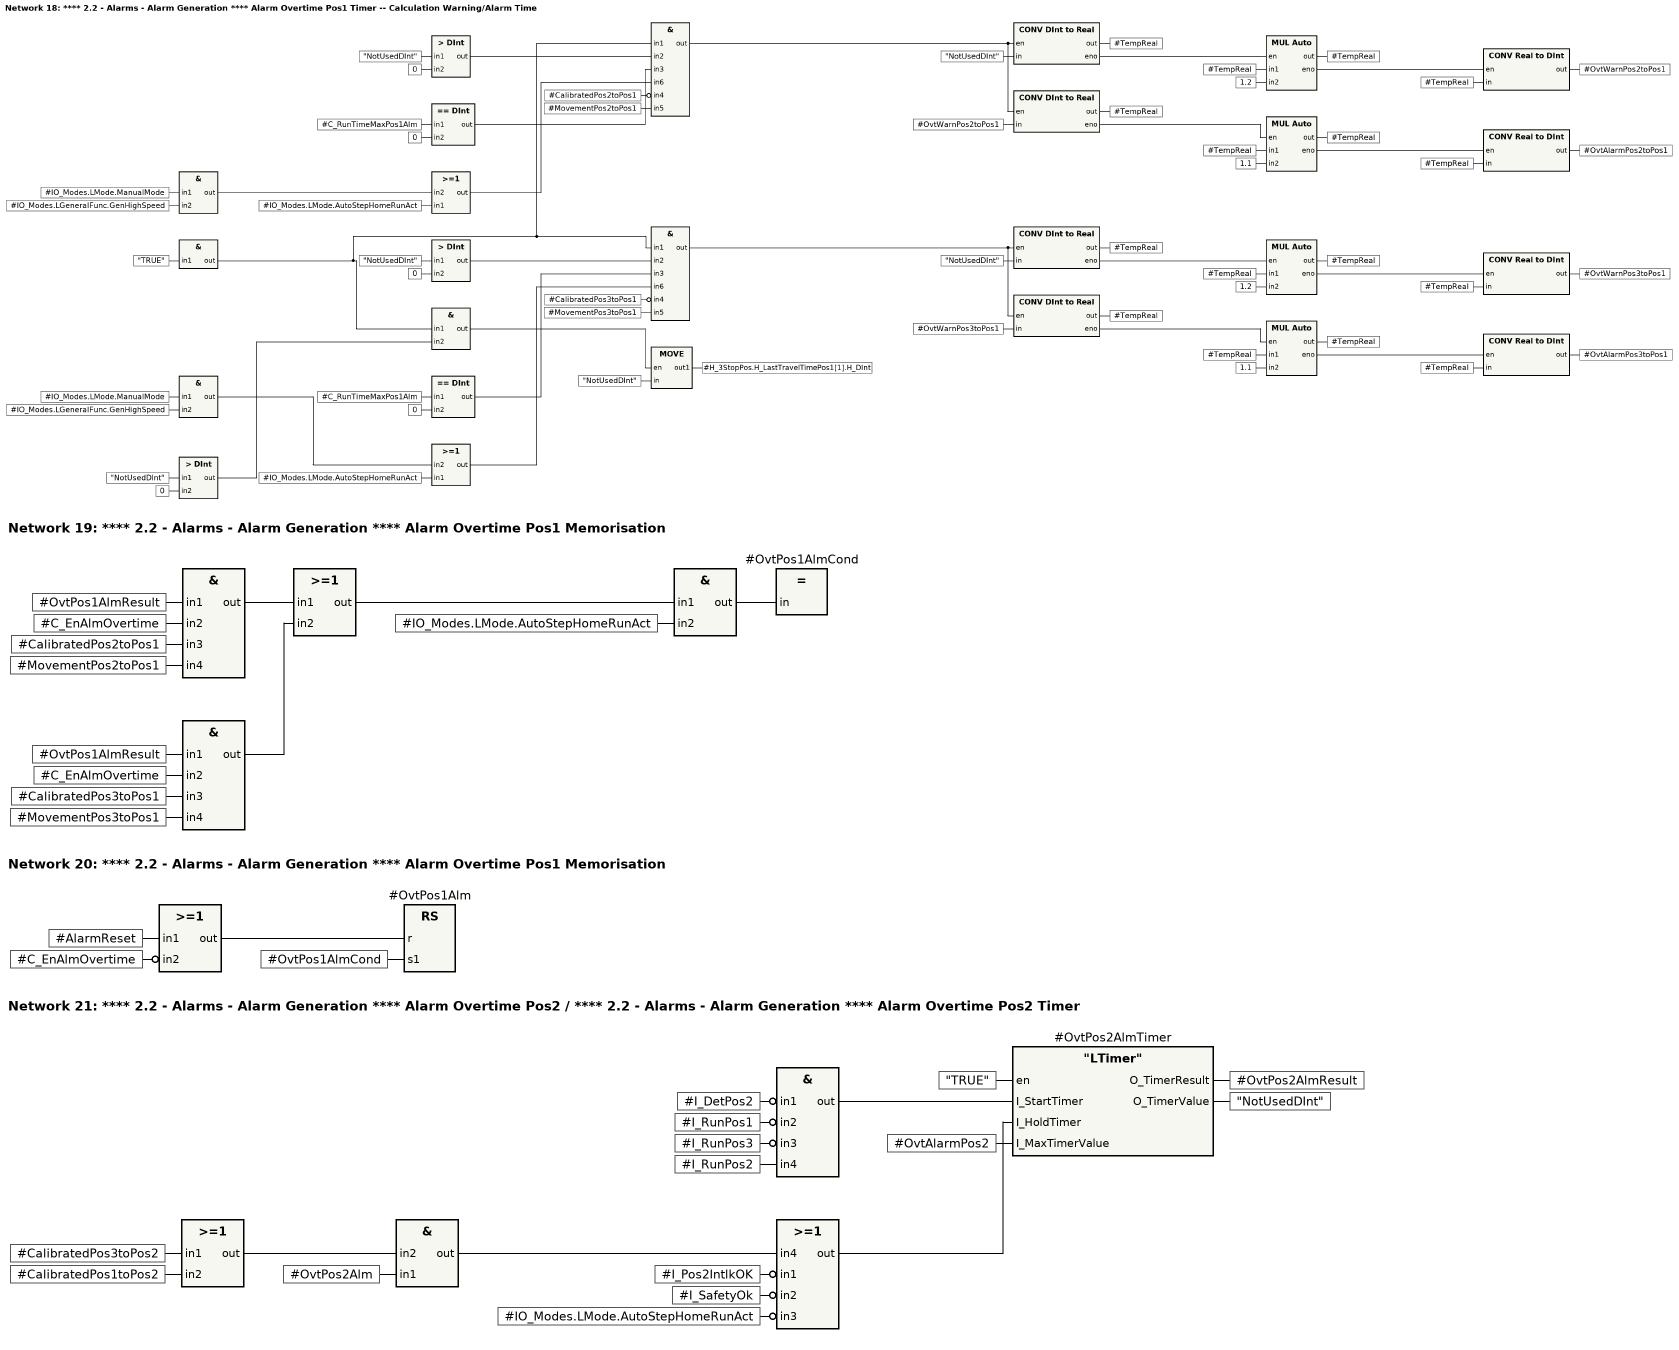
   IF "TRUE" AND ("NotUsedDInt" > 0) AND (#C_RunTimeMaxPos1Alm = 0) AND ((#IO_Modes.LMode.ManualMode AND #IO_Modes.LGeneralFunc.GenHighSpeed) OR #IO_Modes.LMode.AutoStepHomeRunAct) AND NOT #CalibratedPos2toPos1 AND #MovementPos2toPos1 THEN
       #TempReal := DINT_TO_REAL("NotUsedDInt");
       #TempReal := #TempReal * 1.2;
       #OvtWarnPos2toPos1 := REAL_TO_DINT(#TempReal);
       #TempReal := DINT_TO_REAL(#OvtWarnPos2toPos1);
       #TempReal := #TempReal * 1.1;
       #OvtAlarmPos2toPos1 := REAL_TO_DINT(#TempReal);
   END_IF;
   IF "TRUE" AND ("NotUsedDInt" > 0) AND (#C_RunTimeMaxPos1Alm = 0) AND ((#IO_Modes.LMode.ManualMode AND #IO_Modes.LGeneralFunc.GenHighSpeed) OR #IO_Modes.LMode.AutoStepHomeRunAct) AND NOT #CalibratedPos3toPos1 AND #MovementPos3toPos1 THEN
       #TempReal := DINT_TO_REAL("NotUsedDInt");
       #TempReal := #TempReal * 1.2;
       #OvtWarnPos3toPos1 := REAL_TO_DINT(#TempReal);
       #TempReal := DINT_TO_REAL(#OvtWarnPos3toPos1);
       #TempReal := #TempReal * 1.1;
       #OvtAlarmPos3toPos1 := REAL_TO_DINT(#TempReal);
   END_IF;
   IF "TRUE" AND ("NotUsedDInt" > 0) THEN
       #H_3StopPos.H_LastTravelTimePos1[1].H_DInt := "NotUsedDInt";
   END_IF;
END_REGION

REGION Network 19: **** 2.2 - Alarms - Alarm Generation **** Alarm Overtime Pos1 Memorisation
   // Alarm Overtime Pos1 Memorisation
   #OvtPos1AlmCond := ((#OvtPos1AlmResult AND #C_EnAlmOvertime AND #CalibratedPos2toPos1 AND #MovementPos2toPos1) OR (#OvtPos1AlmResult AND #C_EnAlmOvertime AND #CalibratedPos3toPos1 AND #MovementPos3toPos1)) AND #IO_Modes.LMode.AutoStepHomeRunAct;
END_REGION

REGION Network 20: **** 2.2 - Alarms - Alarm Generation **** Alarm Overtime Pos1 Memorisation
   // Alarm Overtime Pos1 Memorisation
   IF #AlarmReset OR NOT #C_EnAlmOvertime THEN
       #OvtPos1Alm := FALSE;   // RS flip-flop
   END_IF;
   IF #OvtPos1AlmCond THEN #OvtPos1Alm := TRUE; END_IF;
END_REGION

REGION Network 21: **** 2.2 - Alarms - Alarm Generation **** Alarm Overtime Pos2 / **** 2.2 - Alarms - Alarm Generation **** Alarm Overtime Pos2 Timer
   // Alarm Overtime Pos2
   IF "TRUE" THEN
       #OvtPos2AlmTimer(I_StartTimer := NOT #I_DetPos2 AND NOT #I_RunPos1 AND NOT #I_RunPos3 AND #I_RunPos2,   // "LTimer"
                        I_HoldTimer := ((#CalibratedPos3toPos2 OR #CalibratedPos1toPos2) AND #OvtPos2Alm) OR NOT #I_Pos2IntlkOK OR NOT #I_SafetyOk OR NOT #IO_Modes.LMode.AutoStepHomeRunAct,
                        I_MaxTimerValue := #OvtAlarmPos2,
                        O_TimerResult => #OvtPos2AlmResult,
                        O_TimerValue => "NotUsedDInt");
   END_IF;
END_REGION

REGION Network 22: **** 2.2 - Alarms - Alarm Generation **** Alarm Overtime Pos2 Timer -- Calculation Warning/Alarm Time
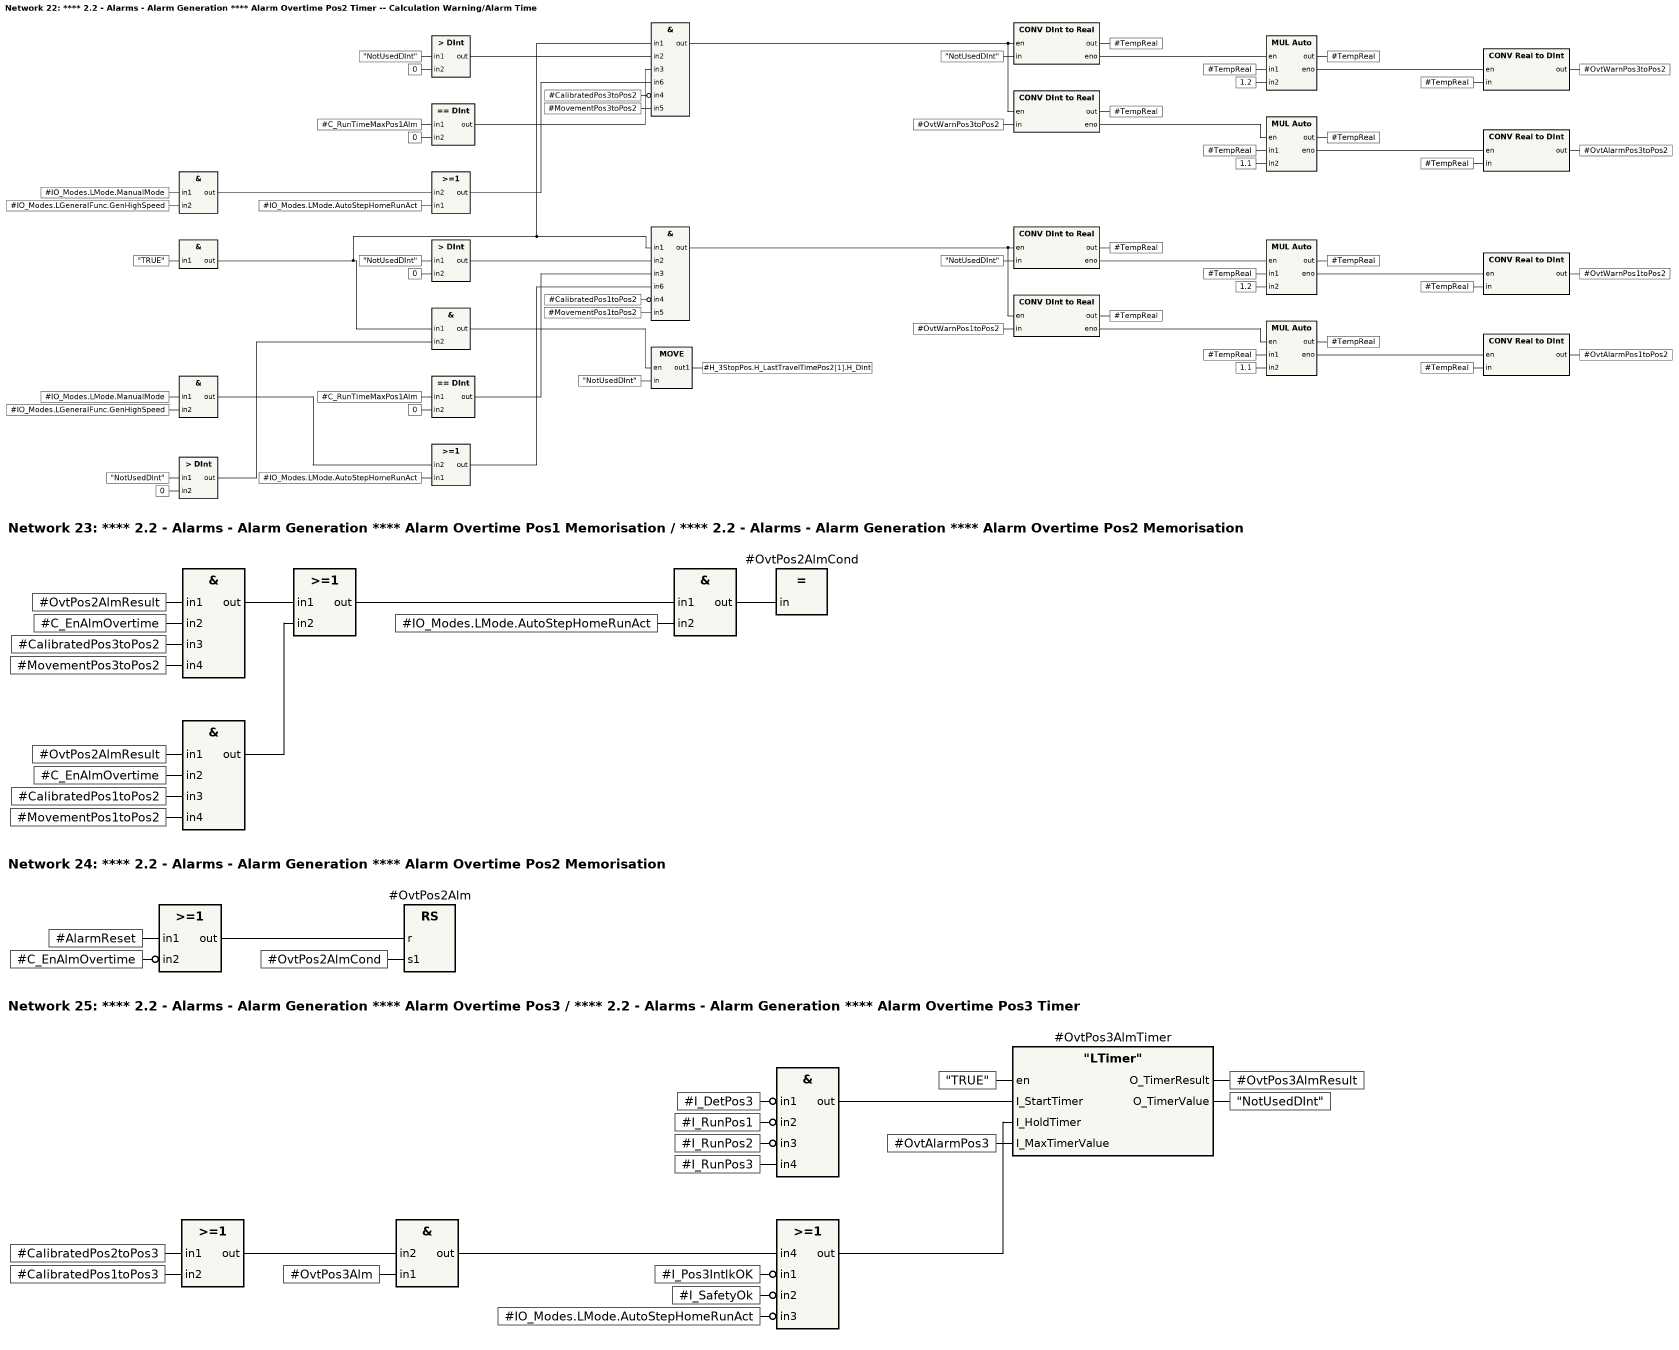
   IF "TRUE" AND ("NotUsedDInt" > 0) AND (#C_RunTimeMaxPos1Alm = 0) AND ((#IO_Modes.LMode.ManualMode AND #IO_Modes.LGeneralFunc.GenHighSpeed) OR #IO_Modes.LMode.AutoStepHomeRunAct) AND NOT #CalibratedPos3toPos2 AND #MovementPos3toPos2 THEN
       #TempReal := DINT_TO_REAL("NotUsedDInt");
       #TempReal := #TempReal * 1.2;
       #OvtWarnPos3toPos2 := REAL_TO_DINT(#TempReal);
       #TempReal := DINT_TO_REAL(#OvtWarnPos3toPos2);
       #TempReal := #TempReal * 1.1;
       #OvtAlarmPos3toPos2 := REAL_TO_DINT(#TempReal);
   END_IF;
   IF "TRUE" AND ("NotUsedDInt" > 0) AND (#C_RunTimeMaxPos1Alm = 0) AND ((#IO_Modes.LMode.ManualMode AND #IO_Modes.LGeneralFunc.GenHighSpeed) OR #IO_Modes.LMode.AutoStepHomeRunAct) AND NOT #CalibratedPos1toPos2 AND #MovementPos1toPos2 THEN
       #TempReal := DINT_TO_REAL("NotUsedDInt");
       #TempReal := #TempReal * 1.2;
       #OvtWarnPos1toPos2 := REAL_TO_DINT(#TempReal);
       #TempReal := DINT_TO_REAL(#OvtWarnPos1toPos2);
       #TempReal := #TempReal * 1.1;
       #OvtAlarmPos1toPos2 := REAL_TO_DINT(#TempReal);
   END_IF;
   IF "TRUE" AND ("NotUsedDInt" > 0) THEN
       #H_3StopPos.H_LastTravelTimePos2[1].H_DInt := "NotUsedDInt";
   END_IF;
END_REGION

REGION Network 23: **** 2.2 - Alarms - Alarm Generation **** Alarm Overtime Pos1 Memorisation / **** 2.2 - Alarms - Alarm Generation **** Alarm Overtime Pos2 Memorisation
   // Alarm Overtime Pos1 Memorisation
   #OvtPos2AlmCond := ((#OvtPos2AlmResult AND #C_EnAlmOvertime AND #CalibratedPos3toPos2 AND #MovementPos3toPos2) OR (#OvtPos2AlmResult AND #C_EnAlmOvertime AND #CalibratedPos1toPos2 AND #MovementPos1toPos2)) AND #IO_Modes.LMode.AutoStepHomeRunAct;
END_REGION

REGION Network 24: **** 2.2 - Alarms - Alarm Generation **** Alarm Overtime Pos2 Memorisation
   // Alarm Overtime Pos2  Memorisation
   IF #AlarmReset OR NOT #C_EnAlmOvertime THEN
       #OvtPos2Alm := FALSE;   // RS flip-flop
   END_IF;
   IF #OvtPos2AlmCond THEN #OvtPos2Alm := TRUE; END_IF;
END_REGION

REGION Network 25: **** 2.2 - Alarms - Alarm Generation **** Alarm Overtime Pos3 / **** 2.2 - Alarms - Alarm Generation **** Alarm Overtime Pos3 Timer
   // Alarm Overtime Pos3
   IF "TRUE" THEN
       #OvtPos3AlmTimer(I_StartTimer := NOT #I_DetPos3 AND NOT #I_RunPos1 AND NOT #I_RunPos2 AND #I_RunPos3,   // "LTimer"
                        I_HoldTimer := ((#CalibratedPos2toPos3 OR #CalibratedPos1toPos3) AND #OvtPos3Alm) OR NOT #I_Pos3IntlkOK OR NOT #I_SafetyOk OR NOT #IO_Modes.LMode.AutoStepHomeRunAct,
                        I_MaxTimerValue := #OvtAlarmPos3,
                        O_TimerResult => #OvtPos3AlmResult,
                        O_TimerValue => "NotUsedDInt");
   END_IF;
END_REGION

REGION Network 26: **** 2.2 - Alarms - Alarm Generation **** Alarm Overtime Pos3 Timer -- Calculation Warning/Alarm Time
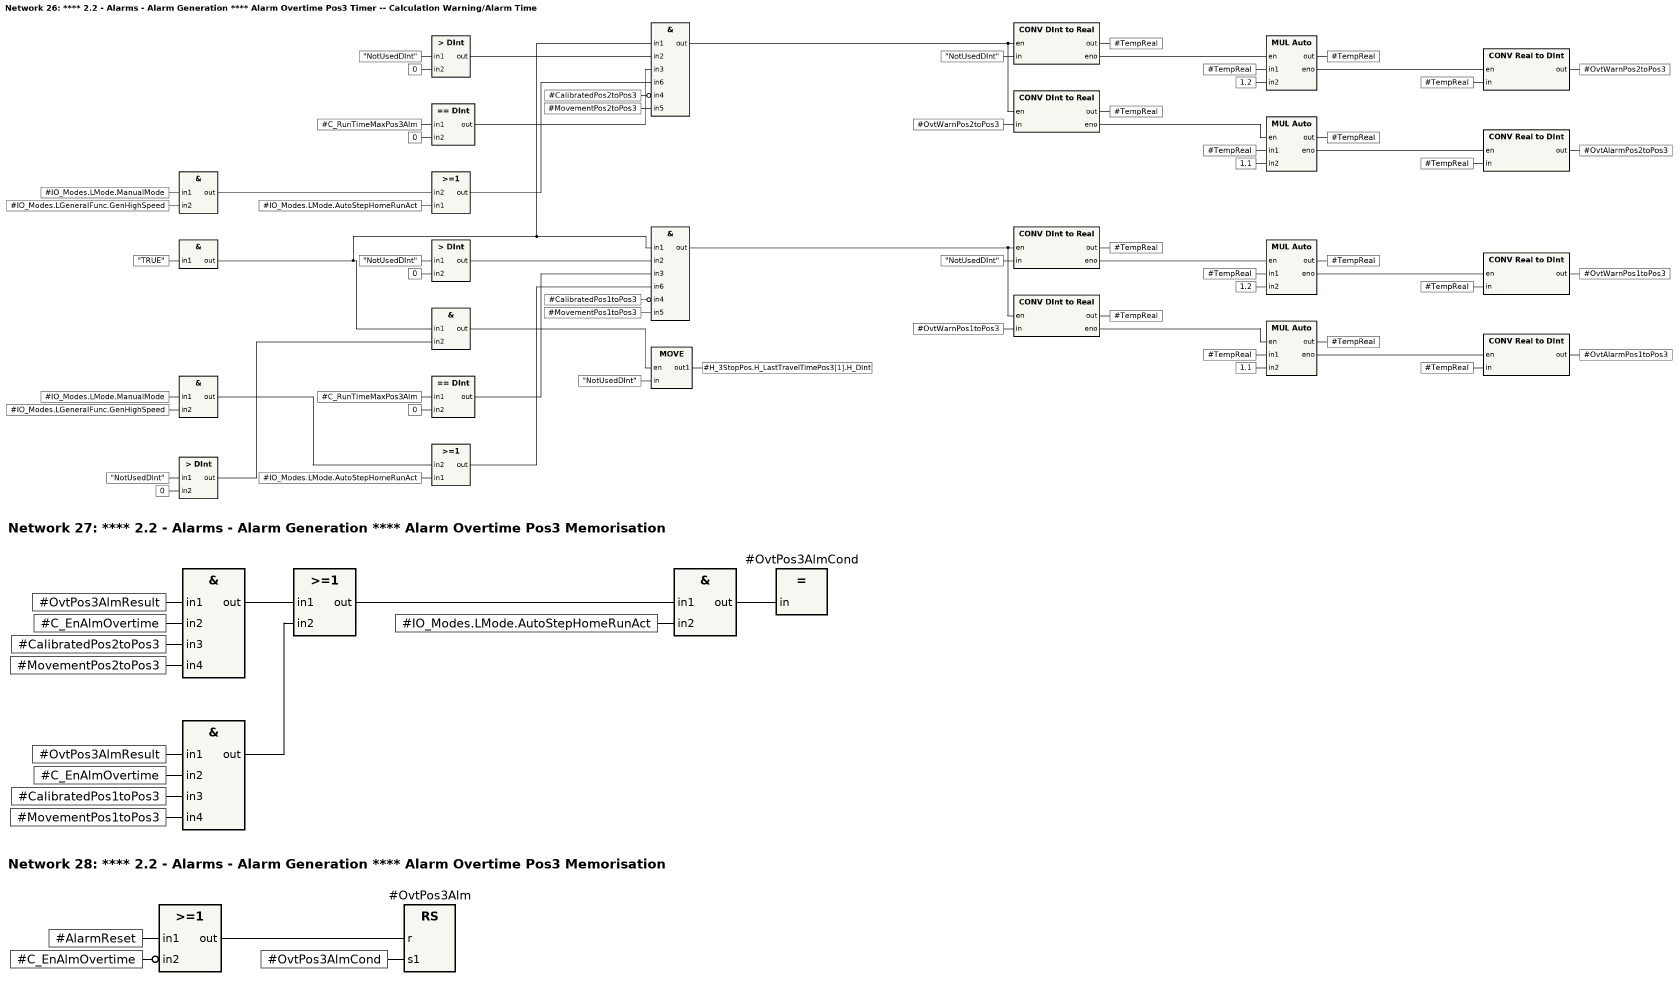
   IF "TRUE" AND ("NotUsedDInt" > 0) AND (#C_RunTimeMaxPos3Alm = 0) AND ((#IO_Modes.LMode.ManualMode AND #IO_Modes.LGeneralFunc.GenHighSpeed) OR #IO_Modes.LMode.AutoStepHomeRunAct) AND NOT #CalibratedPos2toPos3 AND #MovementPos2toPos3 THEN
       #TempReal := DINT_TO_REAL("NotUsedDInt");
       #TempReal := #TempReal * 1.2;
       #OvtWarnPos2toPos3 := REAL_TO_DINT(#TempReal);
       #TempReal := DINT_TO_REAL(#OvtWarnPos2toPos3);
       #TempReal := #TempReal * 1.1;
       #OvtAlarmPos2toPos3 := REAL_TO_DINT(#TempReal);
   END_IF;
   IF "TRUE" AND ("NotUsedDInt" > 0) AND (#C_RunTimeMaxPos3Alm = 0) AND ((#IO_Modes.LMode.ManualMode AND #IO_Modes.LGeneralFunc.GenHighSpeed) OR #IO_Modes.LMode.AutoStepHomeRunAct) AND NOT #CalibratedPos1toPos3 AND #MovementPos1toPos3 THEN
       #TempReal := DINT_TO_REAL("NotUsedDInt");
       #TempReal := #TempReal * 1.2;
       #OvtWarnPos1toPos3 := REAL_TO_DINT(#TempReal);
       #TempReal := DINT_TO_REAL(#OvtWarnPos1toPos3);
       #TempReal := #TempReal * 1.1;
       #OvtAlarmPos1toPos3 := REAL_TO_DINT(#TempReal);
   END_IF;
   IF "TRUE" AND ("NotUsedDInt" > 0) THEN
       #H_3StopPos.H_LastTravelTimePos3[1].H_DInt := "NotUsedDInt";
   END_IF;
END_REGION

REGION Network 27: **** 2.2 - Alarms - Alarm Generation **** Alarm Overtime Pos3 Memorisation
   // Alarm Overtime Pos3  Memorisation
   #OvtPos3AlmCond := ((#OvtPos3AlmResult AND #C_EnAlmOvertime AND #CalibratedPos2toPos3 AND #MovementPos2toPos3) OR (#OvtPos3AlmResult AND #C_EnAlmOvertime AND #CalibratedPos1toPos3 AND #MovementPos1toPos3)) AND #IO_Modes.LMode.AutoStepHomeRunAct;
END_REGION

REGION Network 28: **** 2.2 - Alarms - Alarm Generation **** Alarm Overtime Pos3 Memorisation
   // Alarm Overtime Pos3  Memorisation
   IF #AlarmReset OR NOT #C_EnAlmOvertime THEN
       #OvtPos3Alm := FALSE;   // RS flip-flop
   END_IF;
   IF #OvtPos3AlmCond THEN #OvtPos3Alm := TRUE; END_IF;
END_REGION

REGION Network 29: **** 2.2 - Alarms - Alarm Generation **** Check Amount Of Positions
   // Check Amount Of Positions
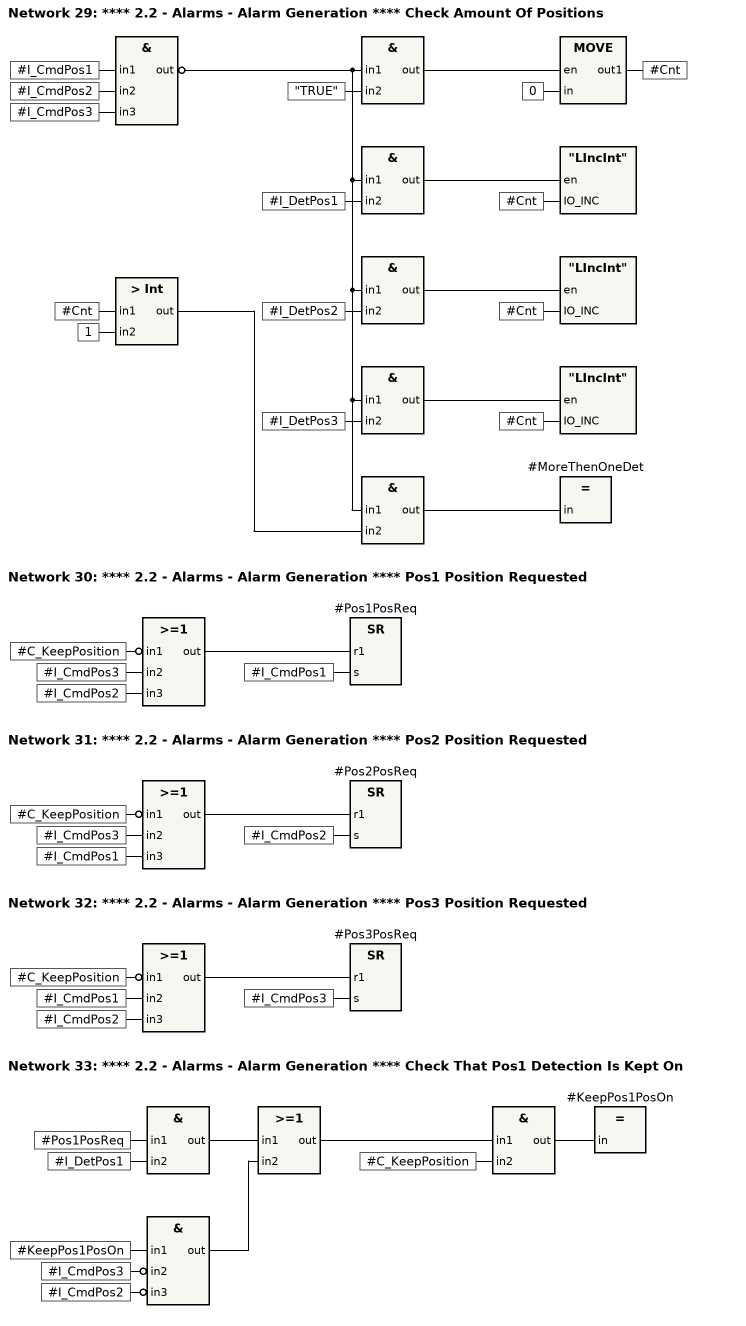
   #_w1 := NOT (#I_CmdPos1 AND #I_CmdPos2 AND #I_CmdPos3);
   IF #_w1 AND "TRUE" THEN #Cnt := 0; END_IF;
   IF #_w1 AND #I_DetPos1 THEN "LIncInt"(IO_INC := #Cnt); END_IF;
   IF #_w1 AND #I_DetPos2 THEN "LIncInt"(IO_INC := #Cnt); END_IF;
   IF #_w1 AND #I_DetPos3 THEN "LIncInt"(IO_INC := #Cnt); END_IF;
   #MoreThenOneDet := #_w1 AND (#Cnt > 1);
END_REGION

REGION Network 30: **** 2.2 - Alarms - Alarm Generation **** Pos1 Position Requested
   // Pos1 Position Requested
   IF #I_CmdPos1 THEN
       #Pos1PosReq := TRUE;   // SR flip-flop
   END_IF;
   IF NOT #C_KeepPosition OR #I_CmdPos3 OR #I_CmdPos2 THEN #Pos1PosReq := FALSE; END_IF;
END_REGION

REGION Network 31: **** 2.2 - Alarms - Alarm Generation **** Pos2 Position Requested
   // Pos2 Position Requested
   IF #I_CmdPos2 THEN
       #Pos2PosReq := TRUE;   // SR flip-flop
   END_IF;
   IF NOT #C_KeepPosition OR #I_CmdPos3 OR #I_CmdPos1 THEN #Pos2PosReq := FALSE; END_IF;
END_REGION

REGION Network 32: **** 2.2 - Alarms - Alarm Generation **** Pos3 Position Requested
   // Pos3  Position Requested
   IF #I_CmdPos3 THEN
       #Pos3PosReq := TRUE;   // SR flip-flop
   END_IF;
   IF NOT #C_KeepPosition OR #I_CmdPos1 OR #I_CmdPos2 THEN #Pos3PosReq := FALSE; END_IF;
END_REGION

REGION Network 33: **** 2.2 - Alarms - Alarm Generation **** Check That Pos1 Detection Is Kept On
   // Check That Pos1 Detection Is Kept On
   #KeepPos1PosOn := ((#Pos1PosReq AND #I_DetPos1) OR (#KeepPos1PosOn AND NOT #I_CmdPos3 AND NOT #I_CmdPos2)) AND #C_KeepPosition;
END_REGION

REGION Network 34: **** 2.2 - Alarms - Alarm Generation **** Check That Pos2 Detection Is Kept On
   // Check That Pos2 Detection Is Kept On
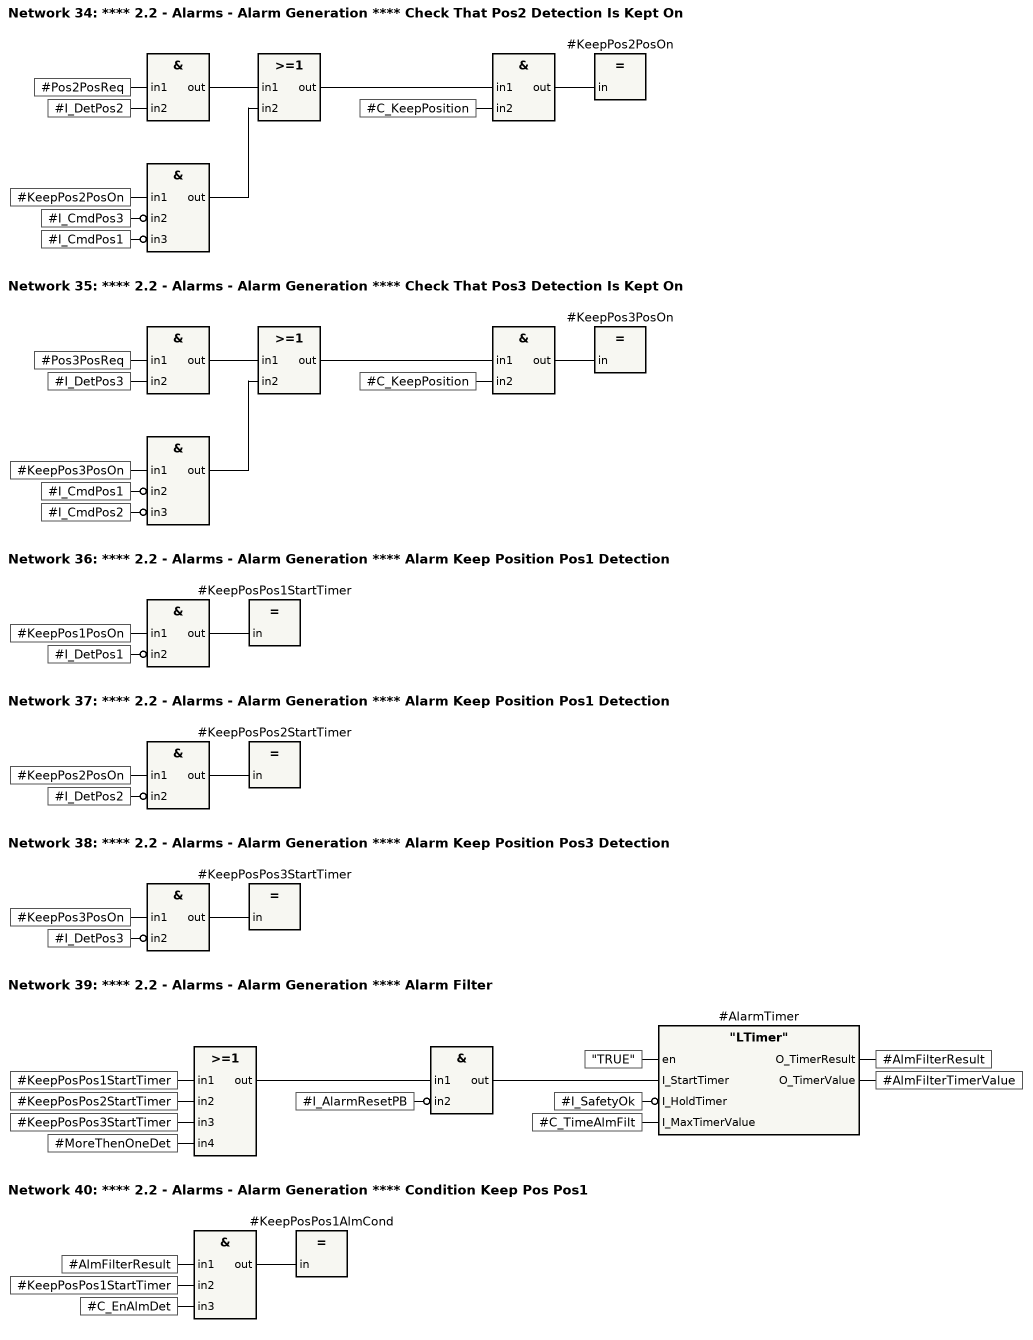
   #KeepPos2PosOn := ((#Pos2PosReq AND #I_DetPos2) OR (#KeepPos2PosOn AND NOT #I_CmdPos3 AND NOT #I_CmdPos1)) AND #C_KeepPosition;
END_REGION

REGION Network 35: **** 2.2 - Alarms - Alarm Generation **** Check That Pos3 Detection Is Kept On
   // Check That Pos3  Detection Is Kept On
   #KeepPos3PosOn := ((#Pos3PosReq AND #I_DetPos3) OR (#KeepPos3PosOn AND NOT #I_CmdPos1 AND NOT #I_CmdPos2)) AND #C_KeepPosition;
END_REGION

REGION Network 36: **** 2.2 - Alarms - Alarm Generation **** Alarm Keep Position Pos1 Detection
   // Alarm keep Position Pos1 Detection
   #KeepPosPos1StartTimer := #KeepPos1PosOn AND NOT #I_DetPos1;
END_REGION

REGION Network 37: **** 2.2 - Alarms - Alarm Generation **** Alarm Keep Position Pos1 Detection
   // Alarm keep Position Pos1 Detection
   #KeepPosPos2StartTimer := #KeepPos2PosOn AND NOT #I_DetPos2;
END_REGION

REGION Network 38: **** 2.2 - Alarms - Alarm Generation **** Alarm Keep Position Pos3 Detection
   // Alarm Keep Position Pos3  Detection
   #KeepPosPos3StartTimer := #KeepPos3PosOn AND NOT #I_DetPos3;
END_REGION

REGION Network 39: **** 2.2 - Alarms - Alarm Generation **** Alarm Filter
   // Alarm Filter
   IF "TRUE" THEN
       #AlarmTimer(I_StartTimer := (#KeepPosPos1StartTimer OR #KeepPosPos2StartTimer OR #KeepPosPos3StartTimer OR #MoreThenOneDet) AND NOT #I_AlarmResetPB,   // "LTimer"
                   I_HoldTimer := NOT #I_SafetyOk,
                   I_MaxTimerValue := #C_TimeAlmFilt,
                   O_TimerResult => #AlmFilterResult,
                   O_TimerValue => #AlmFilterTimerValue);
   END_IF;
END_REGION

REGION Network 40: **** 2.2 - Alarms - Alarm Generation **** Condition Keep Pos Pos1
   // Condition Keep Pos Pos1
   #KeepPosPos1AlmCond := #AlmFilterResult AND #KeepPosPos1StartTimer AND #C_EnAlmDet;
END_REGION

REGION Network 41: **** 2.2 - Alarms - Alarm Generation **** Keep Pos Pos1
   // Keep Pos Pos1
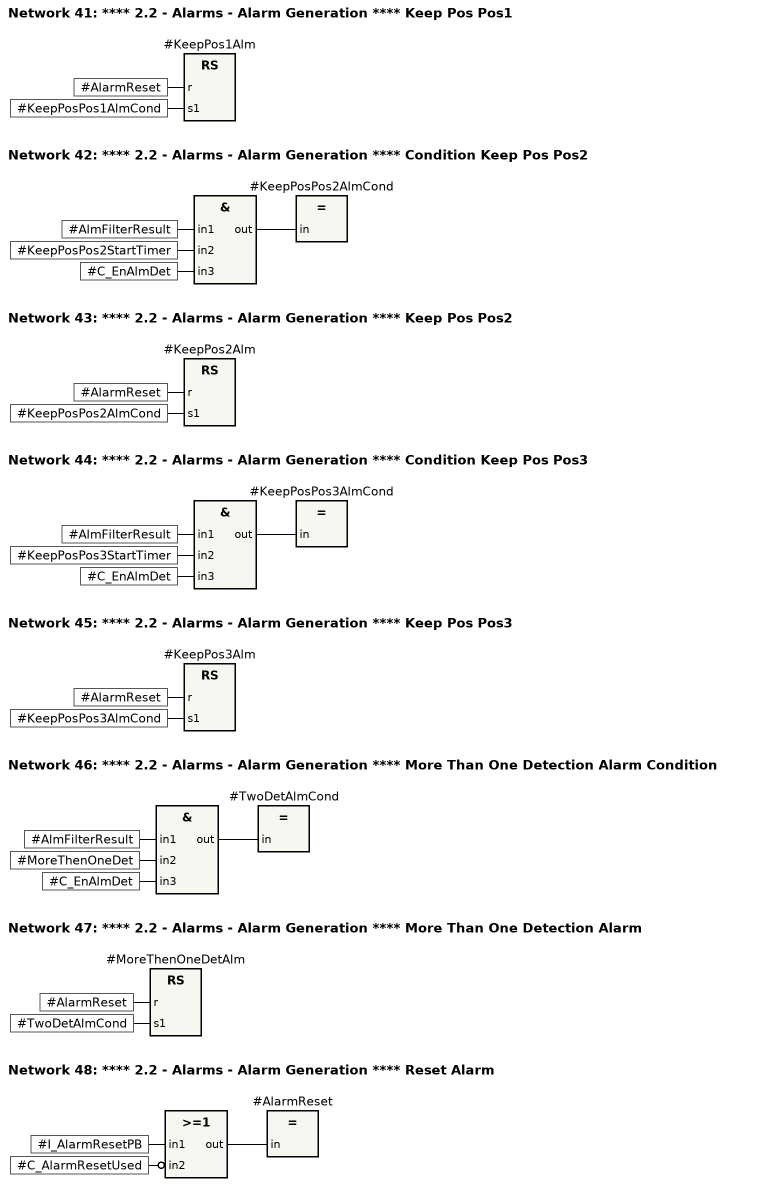
   IF #AlarmReset THEN
       #KeepPos1Alm := FALSE;   // RS flip-flop
   END_IF;
   IF #KeepPosPos1AlmCond THEN #KeepPos1Alm := TRUE; END_IF;
END_REGION

REGION Network 42: **** 2.2 - Alarms - Alarm Generation **** Condition Keep Pos Pos2
   // Condition Keep Pos Pos2
   #KeepPosPos2AlmCond := #AlmFilterResult AND #KeepPosPos2StartTimer AND #C_EnAlmDet;
END_REGION

REGION Network 43: **** 2.2 - Alarms - Alarm Generation **** Keep Pos Pos2
   // Keep Pos Pos2
   IF #AlarmReset THEN
       #KeepPos2Alm := FALSE;   // RS flip-flop
   END_IF;
   IF #KeepPosPos2AlmCond THEN #KeepPos2Alm := TRUE; END_IF;
END_REGION

REGION Network 44: **** 2.2 - Alarms - Alarm Generation **** Condition Keep Pos Pos3
   // Condition Keep Pos Pos3
   #KeepPosPos3AlmCond := #AlmFilterResult AND #KeepPosPos3StartTimer AND #C_EnAlmDet;
END_REGION

REGION Network 45: **** 2.2 - Alarms - Alarm Generation **** Keep Pos Pos3
   // Keep Pos Pos3
   IF #AlarmReset THEN
       #KeepPos3Alm := FALSE;   // RS flip-flop
   END_IF;
   IF #KeepPosPos3AlmCond THEN #KeepPos3Alm := TRUE; END_IF;
END_REGION

REGION Network 46: **** 2.2 - Alarms - Alarm Generation **** More Than One Detection Alarm Condition
   // More Than One Detection Alarm Condition
   #TwoDetAlmCond := #AlmFilterResult AND #MoreThenOneDet AND #C_EnAlmDet;
END_REGION

REGION Network 47: **** 2.2 - Alarms - Alarm Generation **** More Than One Detection Alarm
   // More Than One Detection Alarm
   IF #AlarmReset THEN
       #MoreThenOneDetAlm := FALSE;   // RS flip-flop
   END_IF;
   IF #TwoDetAlmCond THEN #MoreThenOneDetAlm := TRUE; END_IF;
END_REGION

REGION Network 48: **** 2.2 - Alarms - Alarm Generation **** Reset Alarm
   // Reset  Alarm
   #AlarmReset := #I_AlarmResetPB OR NOT #C_AlarmResetUsed;
END_REGION

REGION Network 49: **** 2.2 - Alarms - Alarm Generation **** Config/Calibration Alarm
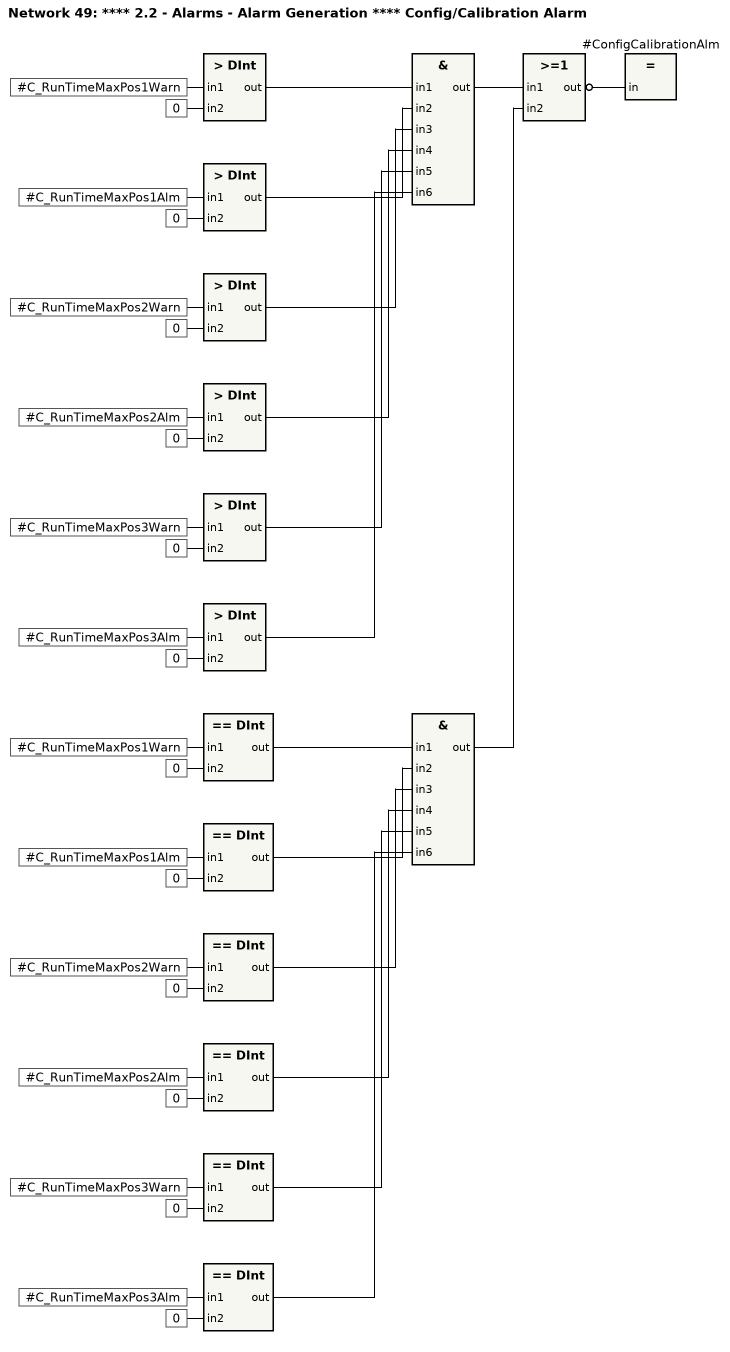
   #ConfigCalibrationAlm := NOT (((#C_RunTimeMaxPos1Warn > 0) AND (#C_RunTimeMaxPos1Alm > 0) AND (#C_RunTimeMaxPos2Warn > 0) AND (#C_RunTimeMaxPos2Alm > 0) AND (#C_RunTimeMaxPos3Warn > 0) AND (#C_RunTimeMaxPos3Alm > 0)) OR ((#C_RunTimeMaxPos1Warn = 0) AND (#C_RunTimeMaxPos1Alm = 0) AND (#C_RunTimeMaxPos2Warn = 0) AND (#C_RunTimeMaxPos2Alm = 0) AND (#C_RunTimeMaxPos3Warn = 0) AND (#C_RunTimeMaxPos3Alm = 0)));
END_REGION

REGION Network 50: **** 2.2 - Alarms - Alarm Generation **** Calibration Warning
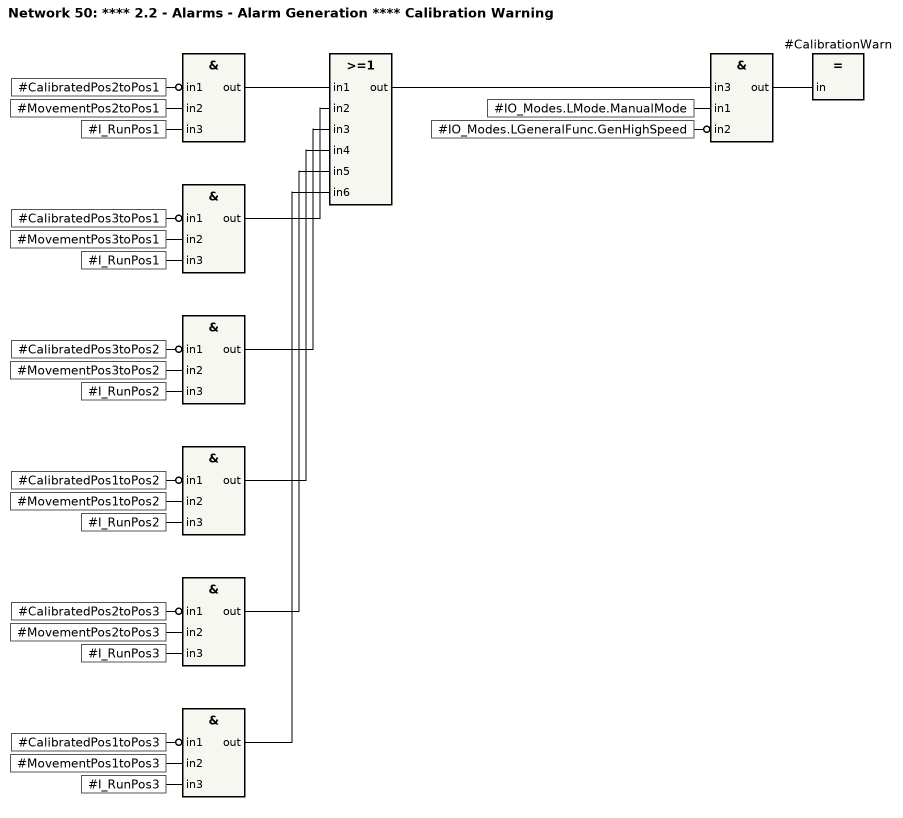
   #CalibrationWarn := ((NOT #CalibratedPos2toPos1 AND #MovementPos2toPos1 AND #I_RunPos1) OR (NOT #CalibratedPos3toPos1 AND #MovementPos3toPos1 AND #I_RunPos1) OR (NOT #CalibratedPos3toPos2 AND #MovementPos3toPos2 AND #I_RunPos2) OR (NOT #CalibratedPos1toPos2 AND #MovementPos1toPos2 AND #I_RunPos2) OR (NOT #CalibratedPos2toPos3 AND #MovementPos2toPos3 AND #I_RunPos3) OR (NOT #CalibratedPos1toPos3 AND #MovementPos1toPos3 AND #I_RunPos3)) AND #IO_Modes.LMode.ManualMode AND NOT #IO_Modes.LGeneralFunc.GenHighSpeed;
END_REGION

REGION Network 51: **** 4.6 - Machine Status - Indication **** Icon Animation
   // Icon Animation
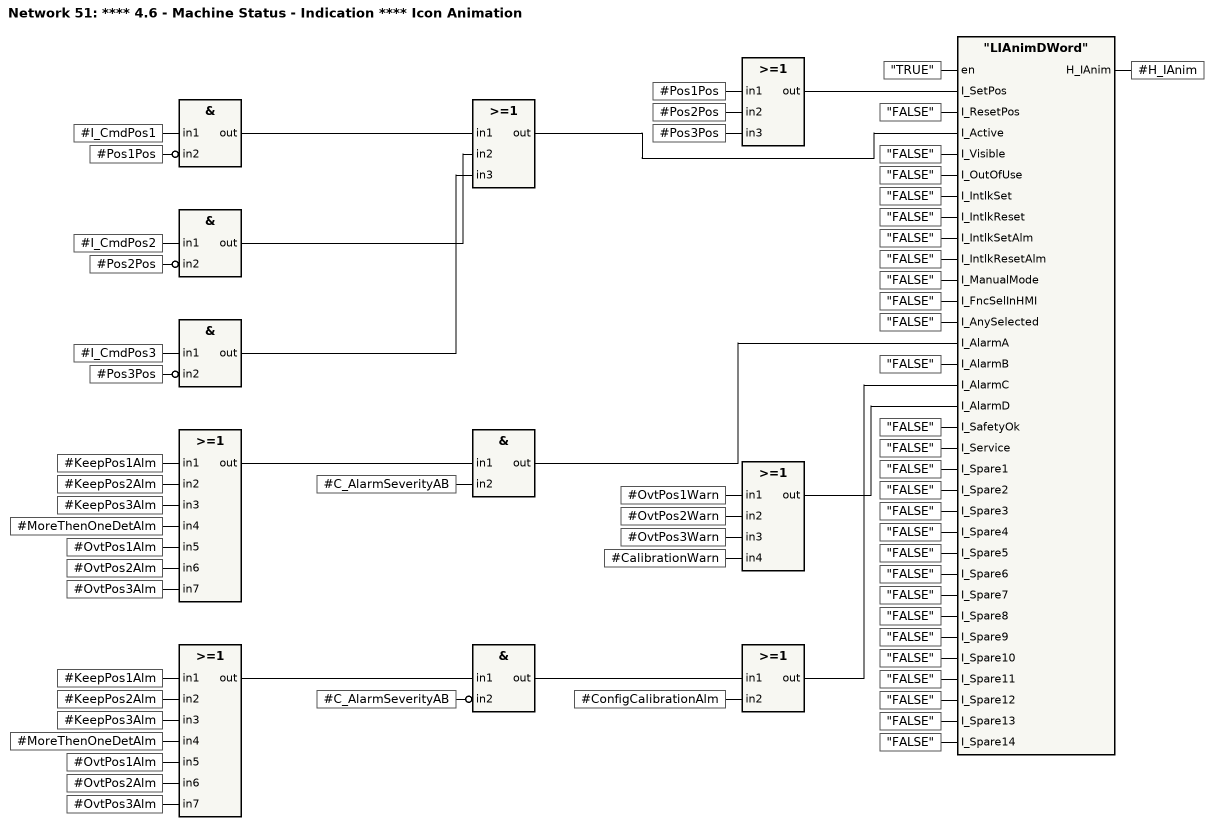
   IF "TRUE" THEN
       "LIAnimDWord"(I_SetPos := #Pos1Pos OR #Pos2Pos OR #Pos3Pos,
                     I_ResetPos := "FALSE",
                     I_Active := (#I_CmdPos1 AND NOT #Pos1Pos) OR (#I_CmdPos2 AND NOT #Pos2Pos) OR (#I_CmdPos3 AND NOT #Pos3Pos),
                     I_Visible := "FALSE",
                     I_OutOfUse := "FALSE",
                     I_IntlkSet := "FALSE",
                     I_IntlkReset := "FALSE",
                     I_IntlkSetAlm := "FALSE",
                     I_IntlkResetAlm := "FALSE",
                     I_ManualMode := "FALSE",
                     I_FncSelInHMI := "FALSE",
                     I_AnySelected := "FALSE",
                     I_AlarmA := (#KeepPos1Alm OR #KeepPos2Alm OR #KeepPos3Alm OR #MoreThenOneDetAlm OR #OvtPos1Alm OR #OvtPos2Alm OR #OvtPos3Alm) AND #C_AlarmSeverityAB,
                     I_AlarmB := "FALSE",
                     I_AlarmC := ((#KeepPos1Alm OR #KeepPos2Alm OR #KeepPos3Alm OR #MoreThenOneDetAlm OR #OvtPos1Alm OR #OvtPos2Alm OR #OvtPos3Alm) AND NOT #C_AlarmSeverityAB) OR #ConfigCalibrationAlm,
                     I_AlarmD := #OvtPos1Warn OR #OvtPos2Warn OR #OvtPos3Warn OR #CalibrationWarn,
                     I_SafetyOk := "FALSE",
                     I_Service := "FALSE",
                     I_Spare1 := "FALSE",
                     I_Spare2 := "FALSE",
                     I_Spare3 := "FALSE",
                     I_Spare4 := "FALSE",
                     I_Spare5 := "FALSE",
                     I_Spare6 := "FALSE",
                     I_Spare7 := "FALSE",
                     I_Spare8 := "FALSE",
                     I_Spare9 := "FALSE",
                     I_Spare10 := "FALSE",
                     I_Spare11 := "FALSE",
                     I_Spare12 := "FALSE",
                     I_Spare13 := "FALSE",
                     I_Spare14 := "FALSE",
                     H_IAnim => #H_IAnim);
   END_IF;
END_REGION

REGION Network 52: **** 4.6 - Machine Status - Indication **** Animation / **** 4.6 - Machine status - Indication **** Animation
   // Animation
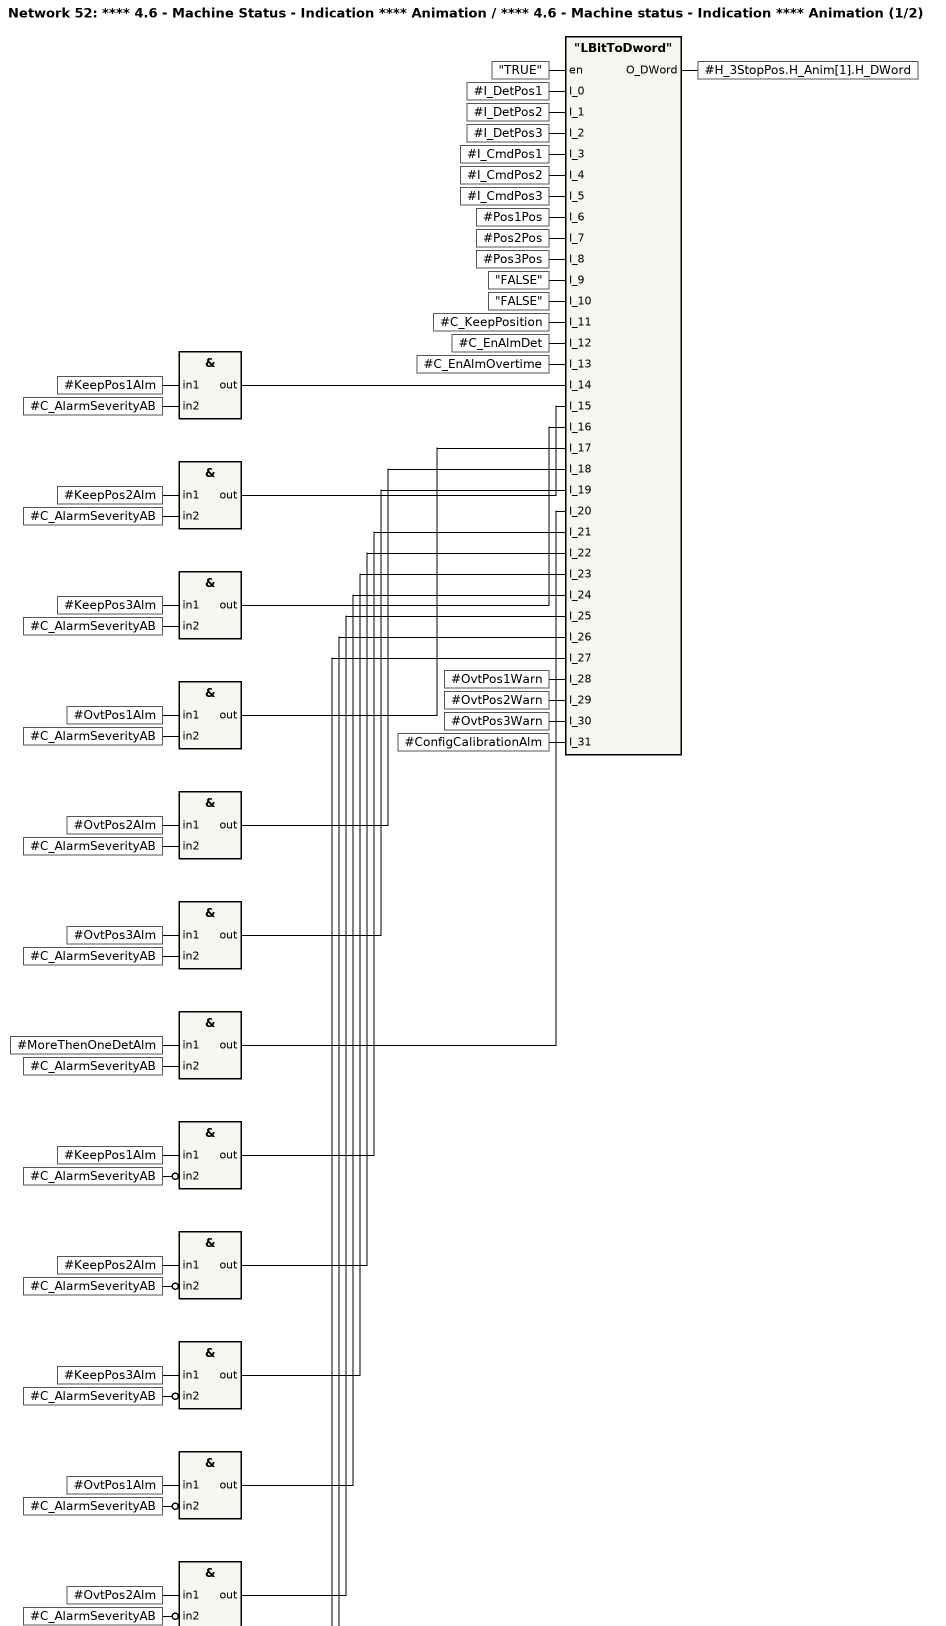
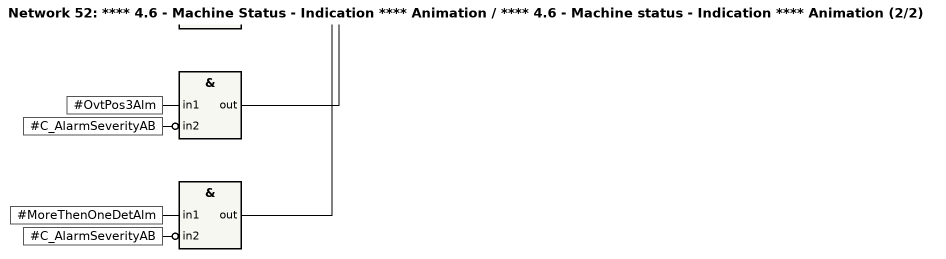
   IF "TRUE" THEN
       "LBitToDword"(I_0 := #I_DetPos1,
                     I_1 := #I_DetPos2,
                     I_2 := #I_DetPos3,
                     I_3 := #I_CmdPos1,
                     I_4 := #I_CmdPos2,
                     I_5 := #I_CmdPos3,
                     I_6 := #Pos1Pos,
                     I_7 := #Pos2Pos,
                     I_8 := #Pos3Pos,
                     I_9 := "FALSE",
                     I_10 := "FALSE",
                     I_11 := #C_KeepPosition,
                     I_12 := #C_EnAlmDet,
                     I_13 := #C_EnAlmOvertime,
                     I_14 := #KeepPos1Alm AND #C_AlarmSeverityAB,
                     I_15 := #KeepPos2Alm AND #C_AlarmSeverityAB,
                     I_16 := #KeepPos3Alm AND #C_AlarmSeverityAB,
                     I_17 := #OvtPos1Alm AND #C_AlarmSeverityAB,
                     I_18 := #OvtPos2Alm AND #C_AlarmSeverityAB,
                     I_19 := #OvtPos3Alm AND #C_AlarmSeverityAB,
                     I_20 := #MoreThenOneDetAlm AND #C_AlarmSeverityAB,
                     I_21 := #KeepPos1Alm AND NOT #C_AlarmSeverityAB,
                     I_22 := #KeepPos2Alm AND NOT #C_AlarmSeverityAB,
                     I_23 := #KeepPos3Alm AND NOT #C_AlarmSeverityAB,
                     I_24 := #OvtPos1Alm AND NOT #C_AlarmSeverityAB,
                     I_25 := #OvtPos2Alm AND NOT #C_AlarmSeverityAB,
                     I_26 := #OvtPos3Alm AND NOT #C_AlarmSeverityAB,
                     I_27 := #MoreThenOneDetAlm AND NOT #C_AlarmSeverityAB,
                     I_28 := #OvtPos1Warn,
                     I_29 := #OvtPos2Warn,
                     I_30 := #OvtPos3Warn,
                     I_31 := #ConfigCalibrationAlm,
                     O_DWord => #H_3StopPos.H_Anim[1].H_DWord);
   END_IF;
END_REGION

REGION Network 53: **** 4.6 - Machine status - Indication **** Animation
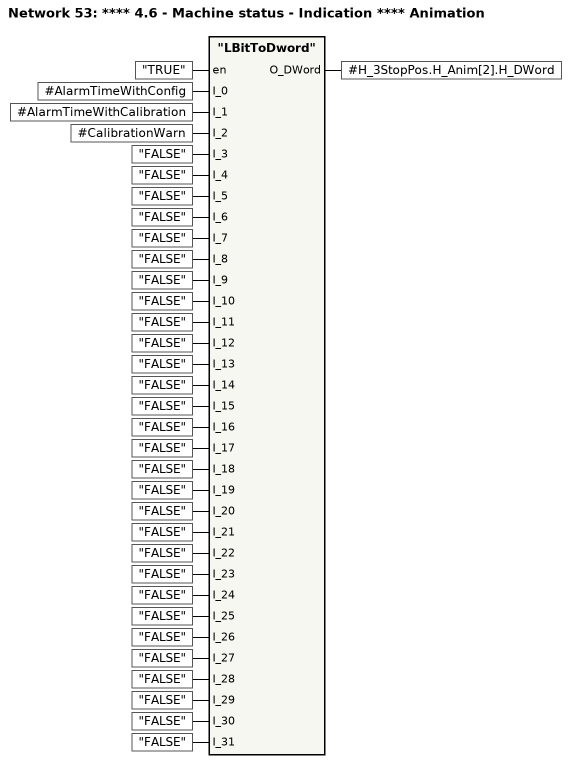
   IF "TRUE" THEN
       "LBitToDword"(I_0 := #AlarmTimeWithConfig,
                     I_1 := #AlarmTimeWithCalibration,
                     I_2 := #CalibrationWarn,
                     I_3 := "FALSE",
                     I_4 := "FALSE",
                     I_5 := "FALSE",
                     I_6 := "FALSE",
                     I_7 := "FALSE",
                     I_8 := "FALSE",
                     I_9 := "FALSE",
                     I_10 := "FALSE",
                     I_11 := "FALSE",
                     I_12 := "FALSE",
                     I_13 := "FALSE",
                     I_14 := "FALSE",
                     I_15 := "FALSE",
                     I_16 := "FALSE",
                     I_17 := "FALSE",
                     I_18 := "FALSE",
                     I_19 := "FALSE",
                     I_20 := "FALSE",
                     I_21 := "FALSE",
                     I_22 := "FALSE",
                     I_23 := "FALSE",
                     I_24 := "FALSE",
                     I_25 := "FALSE",
                     I_26 := "FALSE",
                     I_27 := "FALSE",
                     I_28 := "FALSE",
                     I_29 := "FALSE",
                     I_30 := "FALSE",
                     I_31 := "FALSE",
                     O_DWord => #H_3StopPos.H_Anim[2].H_DWord);
   END_IF;
END_REGION

REGION Network 54: **** 4.6 - Machine status - Indication **** Animation
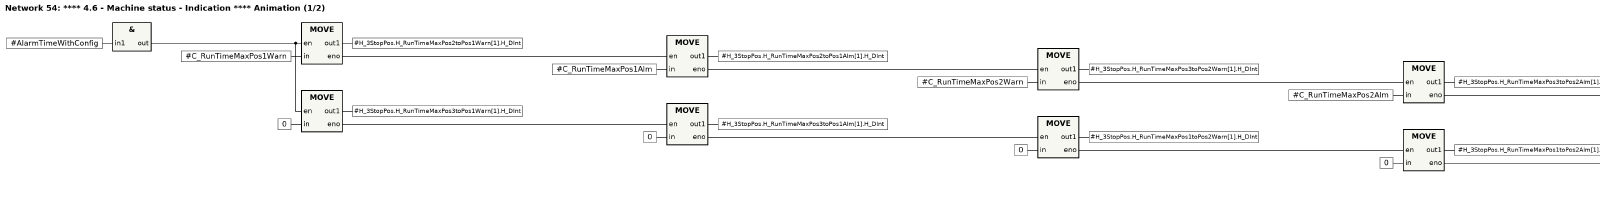
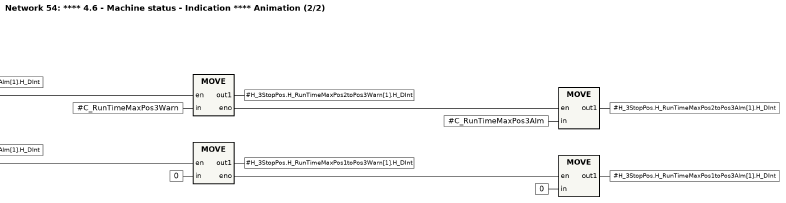
   IF #AlarmTimeWithConfig THEN
       #H_3StopPos.H_RunTimeMaxPos2toPos1Warn[1].H_DInt := #C_RunTimeMaxPos1Warn;
       #H_3StopPos.H_RunTimeMaxPos2toPos1Alm[1].H_DInt := #C_RunTimeMaxPos1Alm;
       #H_3StopPos.H_RunTimeMaxPos3toPos2Warn[1].H_DInt := #C_RunTimeMaxPos2Warn;
       #H_3StopPos.H_RunTimeMaxPos3toPos2Alm[1].H_DInt := #C_RunTimeMaxPos2Alm;
       #H_3StopPos.H_RunTimeMaxPos2toPos3Warn[1].H_DInt := #C_RunTimeMaxPos3Warn;
       #H_3StopPos.H_RunTimeMaxPos2toPos3Alm[1].H_DInt := #C_RunTimeMaxPos3Alm;
       #H_3StopPos.H_RunTimeMaxPos3toPos1Warn[1].H_DInt := 0;
       #H_3StopPos.H_RunTimeMaxPos3toPos1Alm[1].H_DInt := 0;
       #H_3StopPos.H_RunTimeMaxPos1toPos2Warn[1].H_DInt := 0;
       #H_3StopPos.H_RunTimeMaxPos1toPos2Alm[1].H_DInt := 0;
       #H_3StopPos.H_RunTimeMaxPos1toPos3Warn[1].H_DInt := 0;
       #H_3StopPos.H_RunTimeMaxPos1toPos3Alm[1].H_DInt := 0;
   END_IF;
END_REGION

REGION Network 55: **** 4.6 - Machine status - Indication **** Animation
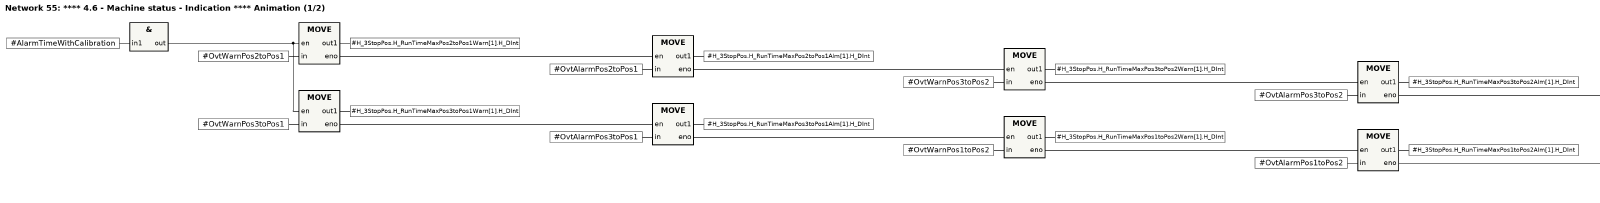
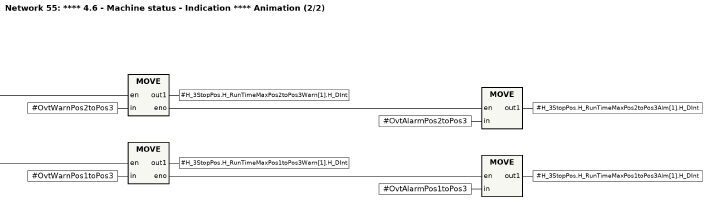
   IF #AlarmTimeWithCalibration THEN
       #H_3StopPos.H_RunTimeMaxPos2toPos1Warn[1].H_DInt := #OvtWarnPos2toPos1;
       #H_3StopPos.H_RunTimeMaxPos2toPos1Alm[1].H_DInt := #OvtAlarmPos2toPos1;
       #H_3StopPos.H_RunTimeMaxPos3toPos2Warn[1].H_DInt := #OvtWarnPos3toPos2;
       #H_3StopPos.H_RunTimeMaxPos3toPos2Alm[1].H_DInt := #OvtAlarmPos3toPos2;
       #H_3StopPos.H_RunTimeMaxPos2toPos3Warn[1].H_DInt := #OvtWarnPos2toPos3;
       #H_3StopPos.H_RunTimeMaxPos2toPos3Alm[1].H_DInt := #OvtAlarmPos2toPos3;
       #H_3StopPos.H_RunTimeMaxPos3toPos1Warn[1].H_DInt := #OvtWarnPos3toPos1;
       #H_3StopPos.H_RunTimeMaxPos3toPos1Alm[1].H_DInt := #OvtAlarmPos3toPos1;
       #H_3StopPos.H_RunTimeMaxPos1toPos2Warn[1].H_DInt := #OvtWarnPos1toPos2;
       #H_3StopPos.H_RunTimeMaxPos1toPos2Alm[1].H_DInt := #OvtAlarmPos1toPos2;
       #H_3StopPos.H_RunTimeMaxPos1toPos3Warn[1].H_DInt := #OvtWarnPos1toPos3;
       #H_3StopPos.H_RunTimeMaxPos1toPos3Alm[1].H_DInt := #OvtAlarmPos1toPos3;
   END_IF;
END_REGION

REGION Network 56: **** 4.6 - Machine status - Indication **** Animation
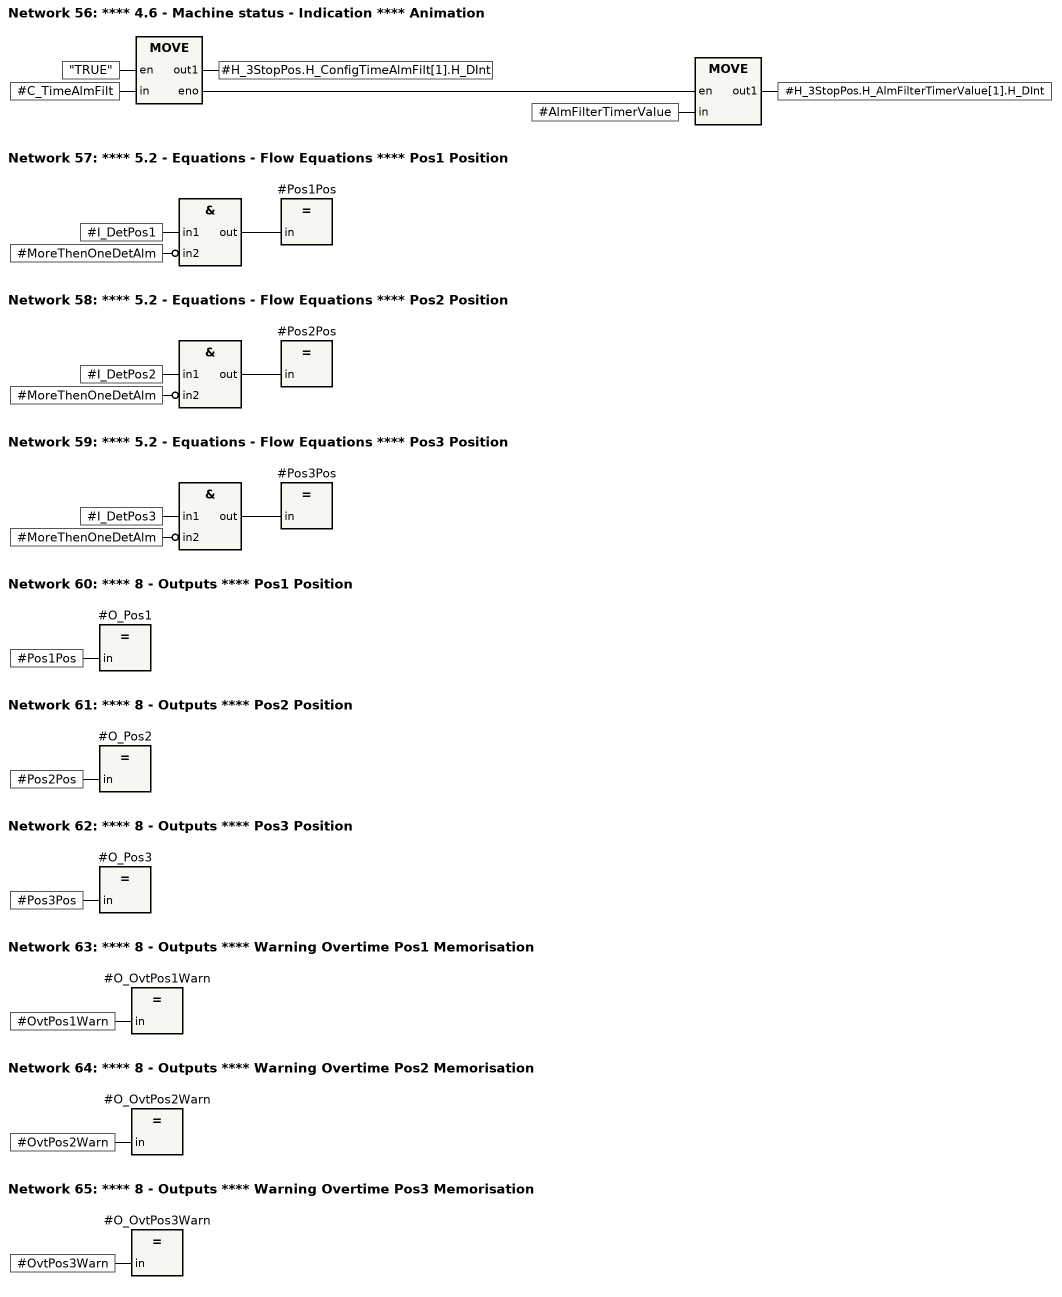
   IF "TRUE" THEN
       #H_3StopPos.H_ConfigTimeAlmFilt[1].H_DInt := #C_TimeAlmFilt;
       #H_3StopPos.H_AlmFilterTimerValue[1].H_DInt := #AlmFilterTimerValue;
   END_IF;
END_REGION

REGION Network 57: **** 5.2 - Equations - Flow Equations **** Pos1 Position
   // Pos1 Position
   #Pos1Pos := #I_DetPos1 AND NOT #MoreThenOneDetAlm;
END_REGION

REGION Network 58: **** 5.2 - Equations - Flow Equations **** Pos2 Position
   // Pos2 Position
   #Pos2Pos := #I_DetPos2 AND NOT #MoreThenOneDetAlm;
END_REGION

REGION Network 59: **** 5.2 - Equations - Flow Equations **** Pos3 Position
   // Pos3  Position
   #Pos3Pos := #I_DetPos3 AND NOT #MoreThenOneDetAlm;
END_REGION

REGION Network 60: **** 8 - Outputs **** Pos1 Position
   // Pos1 Position
   #O_Pos1 := #Pos1Pos;
END_REGION

REGION Network 61: **** 8 - Outputs **** Pos2 Position
   // Pos2 Position
   #O_Pos2 := #Pos2Pos;
END_REGION

REGION Network 62: **** 8 - Outputs **** Pos3 Position
   // Pos3  Position
   #O_Pos3 := #Pos3Pos;
END_REGION

REGION Network 63: **** 8 - Outputs **** Warning Overtime Pos1 Memorisation
   // Warning Overtime Pos1 Memorisation
   #O_OvtPos1Warn := #OvtPos1Warn;
END_REGION

REGION Network 64: **** 8 - Outputs **** Warning Overtime Pos2 Memorisation
   // Warning Overtime Pos2 Memorisation
   #O_OvtPos2Warn := #OvtPos2Warn;
END_REGION

REGION Network 65: **** 8 - Outputs **** Warning Overtime Pos3 Memorisation
   // Warning Overtime Pos3  Memorisation
   #O_OvtPos3Warn := #OvtPos3Warn;
END_REGION

REGION Network 66: **** 8 - Outputs **** Alarm Overtime Pos1 Memorisation
   // Alarm Overtime Pos1 Memorisation
